LIN {X 62.159,Y -33.532,Z -240.496,A -90.000,B 90.000,C 0.000} C_DIS
LIN {X 62.499,Y -33.475,Z -240.051,A -90.000,B 90.000,C 0.000} C_DIS
LIN {X 62.795,Y -33.423,Z -239.682,A -90.000,B 90.000,C 0.000} C_DIS
LIN {X 62.961,Y -33.392,Z -239.489,A -90.000,B 90.000,C 0.000} C_DIS
LIN {X 63.098,Y -33.365,Z -239.345,A -90.000,B 90.000,C 0.000} C_DIS
LIN {X 63.154,Y -33.353,Z -239.294,A -90.000,B 90.000,C 0.000} C_DIS
LIN {X 63.202,Y -33.342,Z -239.257,A -90.000,B 90.000,C 0.000} C_DIS
LIN {X 63.241,Y -33.332,Z -239.236,A -90.000,B 90.000,C 0.000} C_DIS
LIN {X 63.256,Y -33.327,Z -239.231,A -90.000,B 90.000,C 0.000} C_DIS
LIN {X 63.276,Y -33.321,Z -239.232,A -90.000,B 90.000,C 0.000} C_DIS
LIN {X 63.285,Y -33.317,Z -239.238,A -90.000,B 90.000,C 0.000} C_DIS
LIN {X 63.295,Y -33.312,Z -239.255,A -90.000,B 90.000,C 0.000} C_DIS
LIN {X 63.298,Y -33.309,Z -239.272,A -90.000,B 90.000,C 0.000} C_DIS
LIN {X 63.296,Y -33.304,Z -239.320,A -90.000,B 90.000,C 0.000} C_DIS
LIN {X 63.282,Y -33.300,Z -239.387,A -90.000,B 90.000,C 0.000} C_DIS
LIN {X 63.240,Y -33.297,Z -239.526,A -90.000,B 90.000,C 0.000} C_DIS
LIN {X 63.169,Y -33.297,Z -239.713,A -90.000,B 90.000,C 0.000} C_DIS
LIN {X 63.030,Y -33.303,Z -240.041,A -90.000,B 90.000,C 0.000} C_DIS
LIN {X 62.938,Y -33.308,Z -240.240,A -90.000,B 90.000,C 0.000} C_DIS
LIN {X 62.258,Y -33.352,Z -241.702,A -90.000,B 90.000,C 0.000} C_DIS
LIN {X 61.796,Y -33.381,Z -242.689,A -90.000,B 90.000,C 0.000} C_DIS
LIN {X 61.390,Y -33.407,Z -243.561,A -90.000,B 90.000,C 0.000} C_DIS
LIN {X 61.390,Y -60.000,Z -243.561,A -90.000,B 90.000,C 0.000} C_DIS
LIN {X -95.002,Y -60.000,Z -243.561,A -90.000,B 90.000,C 0.000} C_DIS
LIN {X -95.002,Y -34.381,Z -243.561,A -90.000,B 90.000,C 0.000} C_DIS
LIN {X -94.873,Y -34.209,Z -243.260,A -90.000,B 90.000,C 0.000} C_DIS
LIN {X -94.532,Y -34.009,Z -242.776,A -90.000,B 90.000,C 0.000} C_DIS
LIN {X -94.065,Y -33.940,Z -242.365,A -90.000,B 90.000,C 0.000} C_DIS
LIN {X -92.639,Y -33.943,Z -241.367,A -90.000,B 90.000,C 0.000} C_DIS
LIN {X -91.606,Y -33.947,Z -240.642,A -90.000,B 90.000,C 0.000} C_DIS
LIN {X -89.459,Y -33.962,Z -239.147,A -90.000,B 90.000,C 0.000} C_DIS
LIN {X -88.994,Y -33.961,Z -238.830,A -90.000,B 90.000,C 0.000} C_DIS
LIN {X -88.572,Y -33.954,Z -238.548,A -90.000,B 90.000,C 0.000} C_DIS
LIN {X -88.341,Y -33.953,Z -238.396,A -90.000,B 90.000,C 0.000} C_DIS
LIN {X -86.770,Y -33.961,Z -237.376,A -90.000,B 90.000,C 0.000} C_DIS
LIN {X -84.189,Y -33.978,Z -235.700,A -90.000,B 90.000,C 0.000} C_DIS
LIN {X -80.955,Y -34.007,Z -233.615,A -90.000,B 90.000,C 0.000} C_DIS
LIN {X -80.422,Y -34.000,Z -233.284,A -90.000,B 90.000,C 0.000} C_DIS
LIN {X -80.197,Y -33.999,Z -233.147,A -90.000,B 90.000,C 0.000} C_DIS
LIN {X -78.206,Y -34.013,Z -231.959,A -90.000,B 90.000,C 0.000} C_DIS
LIN {X -73.699,Y -34.021,Z -229.309,A -90.000,B 90.000,C 0.000} C_DIS
LIN {X -72.528,Y -34.021,Z -228.623,A -90.000,B 90.000,C 0.000} C_DIS
LIN {X -71.738,Y -34.005,Z -228.177,A -90.000,B 90.000,C 0.000} C_DIS
LIN {X -67.969,Y -34.009,Z -226.154,A -90.000,B 90.000,C 0.000} C_DIS
LIN {X -63.803,Y -34.034,Z -223.947,A -90.000,B 90.000,C 0.000} C_DIS
LIN {X -63.185,Y -34.031,Z -223.626,A -90.000,B 90.000,C 0.000} C_DIS
LIN {X -62.836,Y -34.031,Z -223.448,A -90.000,B 90.000,C 0.000} C_DIS
LIN {X -59.942,Y -34.041,Z -221.989,A -90.000,B 90.000,C 0.000} C_DIS
LIN {X -54.944,Y -34.068,Z -219.481,A -90.000,B 90.000,C 0.000} C_DIS
LIN {X -54.352,Y -34.068,Z -219.187,A -90.000,B 90.000,C 0.000} C_DIS
LIN {X -49.979,Y -34.063,Z -217.035,A -90.000,B 90.000,C 0.000} C_DIS
LIN {X -47.190,Y -34.055,Z -215.668,A -90.000,B 90.000,C 0.000} C_DIS
LIN {X -46.482,Y -34.058,Z -215.318,A -90.000,B 90.000,C 0.000} C_DIS
LIN {X -45.806,Y -34.059,Z -214.980,A -90.000,B 90.000,C 0.000} C_DIS
LIN {X -40.274,Y -34.054,Z -212.247,A -90.000,B 90.000,C 0.000} C_DIS
LIN {X -39.897,Y -34.058,Z -212.057,A -90.000,B 90.000,C 0.000} C_DIS
LIN {X -39.523,Y -34.062,Z -211.867,A -90.000,B 90.000,C 0.000} C_DIS
LIN {X -38.424,Y -34.062,Z -211.295,A -90.000,B 90.000,C 0.000} C_DIS
LIN {X -36.891,Y -34.071,Z -210.490,A -90.000,B 90.000,C 0.000} C_DIS
LIN {X -34.601,Y -34.072,Z -209.269,A -90.000,B 90.000,C 0.000} C_DIS
LIN {X -34.129,Y -34.079,Z -209.011,A -90.000,B 90.000,C 0.000} C_DIS
LIN {X -32.795,Y -34.085,Z -208.262,A -90.000,B 90.000,C 0.000} C_DIS
LIN {X -30.542,Y -34.086,Z -206.982,A -90.000,B 90.000,C 0.000} C_DIS
LIN {X -29.946,Y -34.084,Z -206.646,A -90.000,B 90.000,C 0.000} C_DIS
LIN {X -29.328,Y -34.092,Z -206.286,A -90.000,B 90.000,C 0.000} C_DIS
LIN {X -28.104,Y -34.089,Z -205.541,A -90.000,B 90.000,C 0.000} C_DIS
LIN {X -26.597,Y -34.092,Z -204.635,A -90.000,B 90.000,C 0.000} C_DIS
LIN {X -25.789,Y -34.096,Z -204.147,A -90.000,B 90.000,C 0.000} C_DIS
LIN {X -25.670,Y -34.100,Z -204.073,A -90.000,B 90.000,C 0.000} C_DIS
LIN {X -25.200,Y -34.108,Z -203.778,A -90.000,B 90.000,C 0.000} C_DIS
LIN {X -23.362,Y -34.109,Z -202.572,A -90.000,B 90.000,C 0.000} C_DIS
LIN {X -22.534,Y -34.113,Z -202.026,A -90.000,B 90.000,C 0.000} C_DIS
LIN {X -22.232,Y -34.113,Z -201.824,A -90.000,B 90.000,C 0.000} C_DIS
LIN {X -21.655,Y -34.125,Z -201.428,A -90.000,B 90.000,C 0.000} C_DIS
LIN {X -20.573,Y -34.123,Z -200.645,A -90.000,B 90.000,C 0.000} C_DIS
LIN {X -20.238,Y -34.121,Z -200.404,A -90.000,B 90.000,C 0.000} C_DIS
LIN {X -18.840,Y -34.117,Z -199.408,A -90.000,B 90.000,C 0.000} C_DIS
LIN {X -18.234,Y -34.130,Z -198.963,A -90.000,B 90.000,C 0.000} C_DIS
LIN {X -16.865,Y -34.126,Z -197.899,A -90.000,B 90.000,C 0.000} C_DIS
LIN {X -16.453,Y -34.122,Z -197.581,A -90.000,B 90.000,C 0.000} C_DIS
LIN {X -15.403,Y -34.118,Z -196.780,A -90.000,B 90.000,C 0.000} C_DIS
LIN {X -14.781,Y -34.129,Z -196.292,A -90.000,B 90.000,C 0.000} C_DIS
LIN {X -13.118,Y -34.122,Z -194.933,A -90.000,B 90.000,C 0.000} C_DIS
LIN {X -12.741,Y -34.119,Z -194.626,A -90.000,B 90.000,C 0.000} C_DIS
LIN {X -11.964,Y -34.116,Z -194.000,A -90.000,B 90.000,C 0.000} C_DIS
LIN {X -11.322,Y -34.124,Z -193.473,A -90.000,B 90.000,C 0.000} C_DIS
LIN {X -9.514,Y -34.119,Z -191.943,A -90.000,B 90.000,C 0.000} C_DIS
LIN {X -8.977,Y -34.116,Z -191.491,A -90.000,B 90.000,C 0.000} C_DIS
LIN {X -8.420,Y -34.115,Z -191.025,A -90.000,B 90.000,C 0.000} C_DIS
LIN {X -7.757,Y -34.120,Z -190.465,A -90.000,B 90.000,C 0.000} C_DIS
LIN {X -6.654,Y -34.123,Z -189.524,A -90.000,B 90.000,C 0.000} C_DIS
LIN {X -4.663,Y -34.119,Z -187.811,A -90.000,B 90.000,C 0.000} C_DIS
LIN {X -3.934,Y -34.125,Z -187.175,A -90.000,B 90.000,C 0.000} C_DIS
LIN {X -3.262,Y -34.127,Z -186.589,A -90.000,B 90.000,C 0.000} C_DIS
LIN {X -0.962,Y -34.125,Z -184.573,A -90.000,B 90.000,C 0.000} C_DIS
LIN {X -0.258,Y -34.133,Z -183.947,A -90.000,B 90.000,C 0.000} C_DIS
LIN {X 2.548,Y -34.137,Z -181.427,A -90.000,B 90.000,C 0.000} C_DIS
LIN {X 3.185,Y -34.147,Z -180.848,A -90.000,B 90.000,C 0.000} C_DIS
LIN {X 5.800,Y -34.161,Z -178.421,A -90.000,B 90.000,C 0.000} C_DIS
LIN {X 6.267,Y -34.177,Z -177.976,A -90.000,B 90.000,C 0.000} C_DIS
LIN {X 6.719,Y -34.181,Z -177.529,A -90.000,B 90.000,C 0.000} C_DIS
LIN {X 8.383,Y -34.201,Z -175.896,A -90.000,B 90.000,C 0.000} C_DIS
LIN {X 8.757,Y -34.227,Z -175.511,A -90.000,B 90.000,C 0.000} C_DIS
LIN {X 8.969,Y -34.232,Z -175.270,A -90.000,B 90.000,C 0.000} C_DIS
LIN {X 9.243,Y -34.233,Z -174.965,A -90.000,B 90.000,C 0.000} C_DIS
LIN {X 10.634,Y -34.265,Z -173.481,A -90.000,B 90.000,C 0.000} C_DIS
LIN {X 10.935,Y -34.295,Z -173.139,A -90.000,B 90.000,C 0.000} C_DIS
LIN {X 11.307,Y -34.310,Z -172.649,A -90.000,B 90.000,C 0.000} C_DIS
LIN {X 11.613,Y -34.316,Z -172.255,A -90.000,B 90.000,C 0.000} C_DIS
LIN {X 12.194,Y -34.339,Z -171.552,A -90.000,B 90.000,C 0.000} C_DIS
LIN {X 12.454,Y -34.350,Z -171.236,A -90.000,B 90.000,C 0.000} C_DIS
LIN {X 12.590,Y -34.369,Z -171.060,A -90.000,B 90.000,C 0.000} C_DIS
LIN {X 13.208,Y -34.409,Z -170.063,A -90.000,B 90.000,C 0.000} C_DIS
LIN {X 13.528,Y -34.441,Z -169.537,A -90.000,B 90.000,C 0.000} C_DIS
LIN {X 13.656,Y -34.454,Z -169.331,A -90.000,B 90.000,C 0.000} C_DIS
LIN {X 13.733,Y -34.447,Z -169.124,A -90.000,B 90.000,C 0.000} C_DIS
LIN {X 13.863,Y -34.466,Z -168.731,A -90.000,B 90.000,C 0.000} C_DIS
LIN {X 14.347,Y -34.546,Z -167.346,A -90.000,B 90.000,C 0.000} C_DIS
LIN {X 14.354,Y -34.535,Z -167.206,A -90.000,B 90.000,C 0.000} C_DIS
LIN {X 14.359,Y -34.530,Z -166.963,A -90.000,B 90.000,C 0.000} C_DIS
LIN {X 14.381,Y -34.522,Z -166.386,A -90.000,B 90.000,C 0.000} C_DIS
LIN {X 14.385,Y -34.535,Z -166.076,A -90.000,B 90.000,C 0.000} C_DIS
LIN {X 14.323,Y -34.519,Z -165.696,A -90.000,B 90.000,C 0.000} C_DIS
LIN {X 14.225,Y -34.499,Z -165.096,A -90.000,B 90.000,C 0.000} C_DIS
LIN {X 14.177,Y -34.494,Z -164.732,A -90.000,B 90.000,C 0.000} C_DIS
LIN {X 14.159,Y -34.492,Z -164.583,A -90.000,B 90.000,C 0.000} C_DIS
LIN {X 14.148,Y -34.496,Z -164.509,A -90.000,B 90.000,C 0.000} C_DIS
LIN {X 14.005,Y -34.503,Z -163.900,A -90.000,B 90.000,C 0.000} C_DIS
LIN {X 13.939,Y -34.502,Z -163.607,A -90.000,B 90.000,C 0.000} C_DIS
LIN {X 13.827,Y -34.477,Z -163.300,A -90.000,B 90.000,C 0.000} C_DIS
LIN {X 13.788,Y -34.474,Z -163.199,A -90.000,B 90.000,C 0.000} C_DIS
LIN {X 13.731,Y -34.472,Z -163.029,A -90.000,B 90.000,C 0.000} C_DIS
LIN {X 13.487,Y -34.477,Z -162.191,A -90.000,B 90.000,C 0.000} C_DIS
LIN {X 13.390,Y -34.468,Z -161.928,A -90.000,B 90.000,C 0.000} C_DIS
LIN {X 13.165,Y -34.469,Z -161.344,A -90.000,B 90.000,C 0.000} C_DIS
LIN {X 12.973,Y -34.468,Z -160.825,A -90.000,B 90.000,C 0.000} C_DIS
LIN {X 12.829,Y -34.465,Z -160.458,A -90.000,B 90.000,C 0.000} C_DIS
LIN {X 12.638,Y -34.483,Z -159.999,A -90.000,B 90.000,C 0.000} C_DIS
LIN {X 12.561,Y -34.483,Z -159.848,A -90.000,B 90.000,C 0.000} C_DIS
LIN {X 12.508,Y -34.485,Z -159.739,A -90.000,B 90.000,C 0.000} C_DIS
LIN {X 12.231,Y -34.502,Z -159.117,A -90.000,B 90.000,C 0.000} C_DIS
LIN {X 12.053,Y -34.502,Z -158.705,A -90.000,B 90.000,C 0.000} C_DIS
LIN {X 11.900,Y -34.534,Z -158.371,A -90.000,B 90.000,C 0.000} C_DIS
LIN {X 11.754,Y -34.550,Z -158.111,A -90.000,B 90.000,C 0.000} C_DIS
LIN {X 11.569,Y -34.577,Z -157.758,A -90.000,B 90.000,C 0.000} C_DIS
LIN {X 11.396,Y -34.594,Z -157.422,A -90.000,B 90.000,C 0.000} C_DIS
LIN {X 11.280,Y -34.597,Z -157.187,A -90.000,B 90.000,C 0.000} C_DIS
LIN {X 11.173,Y -34.599,Z -156.961,A -90.000,B 90.000,C 0.000} C_DIS
LIN {X 10.963,Y -34.659,Z -156.564,A -90.000,B 90.000,C 0.000} C_DIS
LIN {X 10.916,Y -34.674,Z -156.471,A -90.000,B 90.000,C 0.000} C_DIS
LIN {X 10.594,Y -34.723,Z -156.014,A -90.000,B 90.000,C 0.000} C_DIS
LIN {X 10.530,Y -34.725,Z -155.919,A -90.000,B 90.000,C 0.000} C_DIS
LIN {X 10.447,Y -34.729,Z -155.796,A -90.000,B 90.000,C 0.000} C_DIS
LIN {X 10.355,Y -34.729,Z -155.658,A -90.000,B 90.000,C 0.000} C_DIS
LIN {X 10.137,Y -34.703,Z -155.488,A -90.000,B 90.000,C 0.000} C_DIS
LIN {X 10.023,Y -34.711,Z -155.408,A -90.000,B 90.000,C 0.000} C_DIS
LIN {X 9.378,Y -34.642,Z -155.286,A -90.000,B 90.000,C 0.000} C_DIS
LIN {X 9.325,Y -34.633,Z -155.286,A -90.000,B 90.000,C 0.000} C_DIS
LIN {X 8.705,Y -34.516,Z -155.315,A -90.000,B 90.000,C 0.000} C_DIS
LIN {X 8.296,Y -34.437,Z -155.335,A -90.000,B 90.000,C 0.000} C_DIS
LIN {X 8.001,Y -34.381,Z -155.347,A -90.000,B 90.000,C 0.000} C_DIS
LIN {X 7.415,Y -34.271,Z -155.366,A -90.000,B 90.000,C 0.000} C_DIS
LIN {X 7.286,Y -34.249,Z -155.365,A -90.000,B 90.000,C 0.000} C_DIS
LIN {X 6.859,Y -34.180,Z -155.350,A -90.000,B 90.000,C 0.000} C_DIS
LIN {X 6.747,Y -34.168,Z -155.347,A -90.000,B 90.000,C 0.000} C_DIS
LIN {X 5.769,Y -34.082,Z -155.287,A -90.000,B 90.000,C 0.000} C_DIS
LIN {X 4.976,Y -34.004,Z -155.251,A -90.000,B 90.000,C 0.000} C_DIS
LIN {X 4.684,Y -33.973,Z -155.233,A -90.000,B 90.000,C 0.000} C_DIS
LIN {X 3.965,Y -33.883,Z -155.172,A -90.000,B 90.000,C 0.000} C_DIS
LIN {X 3.466,Y -33.830,Z -155.115,A -90.000,B 90.000,C 0.000} C_DIS
LIN {X 3.329,Y -33.819,Z -155.094,A -90.000,B 90.000,C 0.000} C_DIS
LIN {X 3.084,Y -33.803,Z -155.049,A -90.000,B 90.000,C 0.000} C_DIS
LIN {X 2.395,Y -33.753,Z -154.935,A -90.000,B 90.000,C 0.000} C_DIS
LIN {X 2.021,Y -33.726,Z -154.871,A -90.000,B 90.000,C 0.000} C_DIS
LIN {X 0.609,Y -33.706,Z -154.731,A -90.000,B 90.000,C 0.000} C_DIS
LIN {X 0.262,Y -33.693,Z -154.684,A -90.000,B 90.000,C 0.000} C_DIS
LIN {X 0.196,Y -33.691,Z -154.674,A -90.000,B 90.000,C 0.000} C_DIS
LIN {X 0.043,Y -33.679,Z -154.641,A -90.000,B 90.000,C 0.000} C_DIS
LIN {X -0.196,Y -33.664,Z -154.586,A -90.000,B 90.000,C 0.000} C_DIS
LIN {X -0.331,Y -33.657,Z -154.551,A -90.000,B 90.000,C 0.000} C_DIS
LIN {X -0.436,Y -33.651,Z -154.524,A -90.000,B 90.000,C 0.000} C_DIS
LIN {X -1.538,Y -33.604,Z -154.234,A -90.000,B 90.000,C 0.000} C_DIS
LIN {X -3.542,Y -33.575,Z -153.793,A -90.000,B 90.000,C 0.000} C_DIS
LIN {X -3.731,Y -33.568,Z -153.746,A -90.000,B 90.000,C 0.000} C_DIS
LIN {X -3.983,Y -33.567,Z -153.678,A -90.000,B 90.000,C 0.000} C_DIS
LIN {X -4.254,Y -33.557,Z -153.585,A -90.000,B 90.000,C 0.000} C_DIS
LIN {X -4.866,Y -33.542,Z -153.370,A -90.000,B 90.000,C 0.000} C_DIS
LIN {X -7.627,Y -33.508,Z -152.461,A -90.000,B 90.000,C 0.000} C_DIS
LIN {X -7.821,Y -33.503,Z -152.386,A -90.000,B 90.000,C 0.000} C_DIS
LIN {X -8.062,Y -33.503,Z -152.291,A -90.000,B 90.000,C 0.000} C_DIS
LIN {X -8.911,Y -33.490,Z -151.916,A -90.000,B 90.000,C 0.000} C_DIS
LIN {X -11.590,Y -33.475,Z -150.786,A -90.000,B 90.000,C 0.000} C_DIS
LIN {X -11.853,Y -33.469,Z -150.658,A -90.000,B 90.000,C 0.000} C_DIS
LIN {X -11.961,Y -33.469,Z -150.604,A -90.000,B 90.000,C 0.000} C_DIS
LIN {X -15.601,Y -33.463,Z -148.685,A -90.000,B 90.000,C 0.000} C_DIS
LIN {X -15.999,Y -33.450,Z -148.437,A -90.000,B 90.000,C 0.000} C_DIS
LIN {X -17.159,Y -33.450,Z -147.679,A -90.000,B 90.000,C 0.000} C_DIS
LIN {X -18.184,Y -33.448,Z -147.012,A -90.000,B 90.000,C 0.000} C_DIS
LIN {X -19.611,Y -33.452,Z -146.104,A -90.000,B 90.000,C 0.000} C_DIS
LIN {X -20.052,Y -33.440,Z -145.768,A -90.000,B 90.000,C 0.000} C_DIS
LIN {X -20.565,Y -33.442,Z -145.372,A -90.000,B 90.000,C 0.000} C_DIS
LIN {X -21.386,Y -33.451,Z -144.756,A -90.000,B 90.000,C 0.000} C_DIS
LIN {X -21.965,Y -33.458,Z -144.321,A -90.000,B 90.000,C 0.000} C_DIS
LIN {X -23.150,Y -33.462,Z -143.408,A -90.000,B 90.000,C 0.000} C_DIS
LIN {X -23.377,Y -33.461,Z -143.227,A -90.000,B 90.000,C 0.000} C_DIS
LIN {X -23.522,Y -33.459,Z -143.110,A -90.000,B 90.000,C 0.000} C_DIS
LIN {X -23.953,Y -33.451,Z -142.721,A -90.000,B 90.000,C 0.000} C_DIS
LIN {X -24.567,Y -33.453,Z -142.160,A -90.000,B 90.000,C 0.000} C_DIS
LIN {X -25.089,Y -33.453,Z -141.686,A -90.000,B 90.000,C 0.000} C_DIS
LIN {X -25.435,Y -33.455,Z -141.379,A -90.000,B 90.000,C 0.000} C_DIS
LIN {X -26.824,Y -33.470,Z -140.144,A -90.000,B 90.000,C 0.000} C_DIS
LIN {X -27.164,Y -33.466,Z -139.812,A -90.000,B 90.000,C 0.000} C_DIS
LIN {X -27.335,Y -33.467,Z -139.632,A -90.000,B 90.000,C 0.000} C_DIS
LIN {X -27.651,Y -33.467,Z -139.290,A -90.000,B 90.000,C 0.000} C_DIS
LIN {X -29.301,Y -33.483,Z -137.499,A -90.000,B 90.000,C 0.000} C_DIS
LIN {X -29.738,Y -33.485,Z -137.021,A -90.000,B 90.000,C 0.000} C_DIS
LIN {X -30.075,Y -33.489,Z -136.657,A -90.000,B 90.000,C 0.000} C_DIS
LIN {X -30.270,Y -33.483,Z -136.415,A -90.000,B 90.000,C 0.000} C_DIS
LIN {X -30.331,Y -33.484,Z -136.338,A -90.000,B 90.000,C 0.000} C_DIS
LIN {X -30.554,Y -33.484,Z -136.043,A -90.000,B 90.000,C 0.000} C_DIS
LIN {X -30.864,Y -33.488,Z -135.631,A -90.000,B 90.000,C 0.000} C_DIS
LIN {X -31.747,Y -33.500,Z -134.465,A -90.000,B 90.000,C 0.000} C_DIS
LIN {X -32.528,Y -33.510,Z -133.429,A -90.000,B 90.000,C 0.000} C_DIS
LIN {X -32.708,Y -33.515,Z -133.188,A -90.000,B 90.000,C 0.000} C_DIS
LIN {X -32.842,Y -33.513,Z -132.986,A -90.000,B 90.000,C 0.000} C_DIS
LIN {X -33.085,Y -33.515,Z -132.587,A -90.000,B 90.000,C 0.000} C_DIS
LIN {X -33.931,Y -33.537,Z -131.182,A -90.000,B 90.000,C 0.000} C_DIS
LIN {X -34.648,Y -33.548,Z -129.959,A -90.000,B 90.000,C 0.000} C_DIS
LIN {X -34.862,Y -33.553,Z -129.592,A -90.000,B 90.000,C 0.000} C_DIS
LIN {X -35.417,Y -33.562,Z -128.408,A -90.000,B 90.000,C 0.000} C_DIS
LIN {X -36.360,Y -33.581,Z -126.392,A -90.000,B 90.000,C 0.000} C_DIS
LIN {X -36.465,Y -33.583,Z -126.158,A -90.000,B 90.000,C 0.000} C_DIS
LIN {X -36.523,Y -33.588,Z -126.023,A -90.000,B 90.000,C 0.000} C_DIS
LIN {X -36.814,Y -33.590,Z -125.230,A -90.000,B 90.000,C 0.000} C_DIS
LIN {X -37.530,Y -33.594,Z -123.280,A -90.000,B 90.000,C 0.000} C_DIS
LIN {X -37.657,Y -33.600,Z -122.924,A -90.000,B 90.000,C 0.000} C_DIS
LIN {X -37.693,Y -33.601,Z -122.812,A -90.000,B 90.000,C 0.000} C_DIS
LIN {X -37.789,Y -33.607,Z -122.510,A -90.000,B 90.000,C 0.000} C_DIS
LIN {X -38.196,Y -33.590,Z -121.049,A -90.000,B 90.000,C 0.000} C_DIS
LIN {X -38.509,Y -33.587,Z -119.908,A -90.000,B 90.000,C 0.000} C_DIS
LIN {X -38.595,Y -33.596,Z -119.573,A -90.000,B 90.000,C 0.000} C_DIS
LIN {X -38.682,Y -33.602,Z -119.190,A -90.000,B 90.000,C 0.000} C_DIS
LIN {X -38.743,Y -33.601,Z -118.872,A -90.000,B 90.000,C 0.000} C_DIS
LIN {X -38.935,Y -33.593,Z -117.837,A -90.000,B 90.000,C 0.000} C_DIS
LIN {X -39.032,Y -33.587,Z -117.334,A -90.000,B 90.000,C 0.000} C_DIS
LIN {X -39.215,Y -33.579,Z -116.390,A -90.000,B 90.000,C 0.000} C_DIS
LIN {X -39.230,Y -33.580,Z -116.307,A -90.000,B 90.000,C 0.000} C_DIS
LIN {X -39.358,Y -33.602,Z -115.575,A -90.000,B 90.000,C 0.000} C_DIS
LIN {X -39.399,Y -33.596,Z -115.225,A -90.000,B 90.000,C 0.000} C_DIS
LIN {X -39.428,Y -33.592,Z -114.983,A -90.000,B 90.000,C 0.000} C_DIS
LIN {X -39.502,Y -33.578,Z -114.284,A -90.000,B 90.000,C 0.000} C_DIS
LIN {X -39.601,Y -33.570,Z -113.300,A -90.000,B 90.000,C 0.000} C_DIS
LIN {X -39.645,Y -33.571,Z -112.836,A -90.000,B 90.000,C 0.000} C_DIS
LIN {X -39.674,Y -33.580,Z -112.458,A -90.000,B 90.000,C 0.000} C_DIS
LIN {X -39.696,Y -33.590,Z -112.185,A -90.000,B 90.000,C 0.000} C_DIS
LIN {X -39.720,Y -33.600,Z -111.769,A -90.000,B 90.000,C 0.000} C_DIS
LIN {X -39.725,Y -33.597,Z -111.269,A -90.000,B 90.000,C 0.000} C_DIS
LIN {X -39.728,Y -33.593,Z -110.998,A -90.000,B 90.000,C 0.000} C_DIS
LIN {X -39.750,Y -33.583,Z -109.970,A -90.000,B 90.000,C 0.000} C_DIS
LIN {X -39.755,Y -33.578,Z -109.563,A -90.000,B 90.000,C 0.000} C_DIS
LIN {X -39.755,Y -33.584,Z -109.062,A -90.000,B 90.000,C 0.000} C_DIS
LIN {X -39.755,Y -33.585,Z -109.015,A -90.000,B 90.000,C 0.000} C_DIS
LIN {X -39.752,Y -33.601,Z -108.594,A -90.000,B 90.000,C 0.000} C_DIS
LIN {X -39.738,Y -33.617,Z -108.151,A -90.000,B 90.000,C 0.000} C_DIS
LIN {X -39.618,Y -33.621,Z -106.728,A -90.000,B 90.000,C 0.000} C_DIS
LIN {X -39.591,Y -33.630,Z -106.282,A -90.000,B 90.000,C 0.000} C_DIS
LIN {X -39.570,Y -33.641,Z -105.984,A -90.000,B 90.000,C 0.000} C_DIS
LIN {X -39.574,Y -33.649,Z -105.933,A -90.000,B 90.000,C 0.000} C_DIS
LIN {X -39.603,Y -33.689,Z -105.733,A -90.000,B 90.000,C 0.000} C_DIS
LIN {X -39.687,Y -33.905,Z -104.786,A -90.000,B 90.000,C 0.000} C_DIS
LIN {X -39.703,Y -33.985,Z -104.461,A -90.000,B 90.000,C 0.000} C_DIS
LIN {X -39.715,Y -34.034,Z -104.290,A -90.000,B 90.000,C 0.000} C_DIS
LIN {X -39.730,Y -34.114,Z -104.019,A -90.000,B 90.000,C 0.000} C_DIS
LIN {X -39.737,Y -34.256,Z -103.511,A -90.000,B 90.000,C 0.000} C_DIS
LIN {X -39.735,Y -34.336,Z -103.233,A -90.000,B 90.000,C 0.000} C_DIS
LIN {X -39.728,Y -34.377,Z -103.097,A -90.000,B 90.000,C 0.000} C_DIS
LIN {X -39.716,Y -34.428,Z -102.932,A -90.000,B 90.000,C 0.000} C_DIS
LIN {X -39.687,Y -34.522,Z -102.629,A -90.000,B 90.000,C 0.000} C_DIS
LIN {X -39.794,Y -34.529,Z -102.461,A -90.000,B 90.000,C 0.000} C_DIS
LIN {X -39.978,Y -34.527,Z -102.218,A -90.000,B 90.000,C 0.000} C_DIS
LIN {X -40.274,Y -34.520,Z -101.825,A -90.000,B 90.000,C 0.000} C_DIS
LIN {X -40.484,Y -34.518,Z -101.540,A -90.000,B 90.000,C 0.000} C_DIS
LIN {X -40.926,Y -34.522,Z -100.945,A -90.000,B 90.000,C 0.000} C_DIS
LIN {X -41.149,Y -34.528,Z -100.633,A -90.000,B 90.000,C 0.000} C_DIS
LIN {X -41.594,Y -34.528,Z -99.995,A -90.000,B 90.000,C 0.000} C_DIS
LIN {X -41.989,Y -34.521,Z -99.424,A -90.000,B 90.000,C 0.000} C_DIS
LIN {X -42.209,Y -34.519,Z -99.094,A -90.000,B 90.000,C 0.000} C_DIS
LIN {X -43.182,Y -34.537,Z -97.528,A -90.000,B 90.000,C 0.000} C_DIS
LIN {X -43.779,Y -34.537,Z -96.531,A -90.000,B 90.000,C 0.000} C_DIS
LIN {X -44.127,Y -34.542,Z -95.910,A -90.000,B 90.000,C 0.000} C_DIS
LIN {X -44.243,Y -34.545,Z -95.693,A -90.000,B 90.000,C 0.000} C_DIS
LIN {X -44.690,Y -34.548,Z -94.867,A -90.000,B 90.000,C 0.000} C_DIS
LIN {X -45.006,Y -34.543,Z -94.279,A -90.000,B 90.000,C 0.000} C_DIS
LIN {X -45.634,Y -34.529,Z -93.045,A -90.000,B 90.000,C 0.000} C_DIS
LIN {X -45.784,Y -34.527,Z -92.725,A -90.000,B 90.000,C 0.000} C_DIS
LIN {X -45.928,Y -34.524,Z -92.409,A -90.000,B 90.000,C 0.000} C_DIS
LIN {X -46.226,Y -34.527,Z -91.706,A -90.000,B 90.000,C 0.000} C_DIS
LIN {X -46.345,Y -34.531,Z -91.429,A -90.000,B 90.000,C 0.000} C_DIS
LIN {X -46.588,Y -34.531,Z -90.852,A -90.000,B 90.000,C 0.000} C_DIS
LIN {X -46.672,Y -34.529,Z -90.650,A -90.000,B 90.000,C 0.000} C_DIS
LIN {X -46.795,Y -34.524,Z -90.342,A -90.000,B 90.000,C 0.000} C_DIS
LIN {X -47.062,Y -34.518,Z -89.640,A -90.000,B 90.000,C 0.000} C_DIS
LIN {X -47.276,Y -34.515,Z -89.066,A -90.000,B 90.000,C 0.000} C_DIS
LIN {X -47.307,Y -34.515,Z -88.976,A -90.000,B 90.000,C 0.000} C_DIS
LIN {X -47.481,Y -34.521,Z -88.439,A -90.000,B 90.000,C 0.000} C_DIS
LIN {X -47.708,Y -34.530,Z -87.635,A -90.000,B 90.000,C 0.000} C_DIS
LIN {X -47.958,Y -34.555,Z -86.619,A -90.000,B 90.000,C 0.000} C_DIS
LIN {X -48.119,Y -34.563,Z -85.944,A -90.000,B 90.000,C 0.000} C_DIS
LIN {X -48.237,Y -34.565,Z -85.444,A -90.000,B 90.000,C 0.000} C_DIS
LIN {X -48.290,Y -34.565,Z -85.230,A -90.000,B 90.000,C 0.000} C_DIS
LIN {X -48.318,Y -34.563,Z -85.110,A -90.000,B 90.000,C 0.000} C_DIS
LIN {X -48.354,Y -34.562,Z -84.920,A -90.000,B 90.000,C 0.000} C_DIS
LIN {X -48.399,Y -34.567,Z -84.609,A -90.000,B 90.000,C 0.000} C_DIS
LIN {X -48.445,Y -34.574,Z -84.247,A -90.000,B 90.000,C 0.000} C_DIS
LIN {X -48.490,Y -34.586,Z -83.828,A -90.000,B 90.000,C 0.000} C_DIS
LIN {X -48.573,Y -34.613,Z -83.086,A -90.000,B 90.000,C 0.000} C_DIS
LIN {X -48.605,Y -34.616,Z -82.769,A -90.000,B 90.000,C 0.000} C_DIS
LIN {X -48.642,Y -34.615,Z -82.371,A -90.000,B 90.000,C 0.000} C_DIS
LIN {X -48.646,Y -34.620,Z -82.172,A -90.000,B 90.000,C 0.000} C_DIS
LIN {X -48.616,Y -34.663,Z -81.147,A -90.000,B 90.000,C 0.000} C_DIS
LIN {X -48.606,Y -34.674,Z -80.924,A -90.000,B 90.000,C 0.000} C_DIS
LIN {X -48.552,Y -34.680,Z -79.949,A -90.000,B 90.000,C 0.000} C_DIS
LIN {X -48.532,Y -34.685,Z -79.752,A -90.000,B 90.000,C 0.000} C_DIS
LIN {X -48.441,Y -34.707,Z -79.153,A -90.000,B 90.000,C 0.000} C_DIS
LIN {X -48.394,Y -34.717,Z -78.846,A -90.000,B 90.000,C 0.000} C_DIS
LIN {X -48.360,Y -34.721,Z -78.650,A -90.000,B 90.000,C 0.000} C_DIS
LIN {X -48.232,Y -34.730,Z -77.986,A -90.000,B 90.000,C 0.000} C_DIS
LIN {X -48.159,Y -34.735,Z -77.625,A -90.000,B 90.000,C 0.000} C_DIS
LIN {X -48.134,Y -34.738,Z -77.513,A -90.000,B 90.000,C 0.000} C_DIS
LIN {X -47.991,Y -34.754,Z -76.959,A -90.000,B 90.000,C 0.000} C_DIS
LIN {X -47.818,Y -34.767,Z -76.298,A -90.000,B 90.000,C 0.000} C_DIS
LIN {X -47.774,Y -34.768,Z -76.136,A -90.000,B 90.000,C 0.000} C_DIS
LIN {X -47.689,Y -34.771,Z -75.857,A -90.000,B 90.000,C 0.000} C_DIS
LIN {X -47.567,Y -34.777,Z -75.486,A -90.000,B 90.000,C 0.000} C_DIS
LIN {X -47.263,Y -34.794,Z -74.623,A -90.000,B 90.000,C 0.000} C_DIS
LIN {X -47.123,Y -34.795,Z -74.230,A -90.000,B 90.000,C 0.000} C_DIS
LIN {X -47.075,Y -34.796,Z -74.107,A -90.000,B 90.000,C 0.000} C_DIS
LIN {X -46.850,Y -34.804,Z -73.585,A -90.000,B 90.000,C 0.000} C_DIS
LIN {X -46.642,Y -34.812,Z -73.094,A -90.000,B 90.000,C 0.000} C_DIS
LIN {X -46.444,Y -34.811,Z -72.632,A -90.000,B 90.000,C 0.000} C_DIS
LIN {X -46.371,Y -34.812,Z -72.477,A -90.000,B 90.000,C 0.000} C_DIS
LIN {X -46.171,Y -34.817,Z -72.066,A -90.000,B 90.000,C 0.000} C_DIS
LIN {X -46.140,Y -34.816,Z -72.004,A -90.000,B 90.000,C 0.000} C_DIS
LIN {X -45.985,Y -34.817,Z -71.720,A -90.000,B 90.000,C 0.000} C_DIS
LIN {X -45.865,Y -34.818,Z -71.518,A -90.000,B 90.000,C 0.000} C_DIS
LIN {X -45.457,Y -34.816,Z -70.840,A -90.000,B 90.000,C 0.000} C_DIS
LIN {X -45.413,Y -34.817,Z -70.771,A -90.000,B 90.000,C 0.000} C_DIS
LIN {X -45.178,Y -34.820,Z -70.412,A -90.000,B 90.000,C 0.000} C_DIS
LIN {X -44.948,Y -34.806,Z -70.070,A -90.000,B 90.000,C 0.000} C_DIS
LIN {X -44.890,Y -34.803,Z -69.989,A -90.000,B 90.000,C 0.000} C_DIS
LIN {X -44.795,Y -34.800,Z -69.873,A -90.000,B 90.000,C 0.000} C_DIS
LIN {X -44.594,Y -34.796,Z -69.646,A -90.000,B 90.000,C 0.000} C_DIS
LIN {X -44.093,Y -34.796,Z -69.111,A -90.000,B 90.000,C 0.000} C_DIS
LIN {X -43.839,Y -34.796,Z -68.858,A -90.000,B 90.000,C 0.000} C_DIS
LIN {X -43.669,Y -34.786,Z -68.693,A -90.000,B 90.000,C 0.000} C_DIS
LIN {X -43.172,Y -34.748,Z -68.214,A -90.000,B 90.000,C 0.000} C_DIS
LIN {X -42.967,Y -34.737,Z -68.041,A -90.000,B 90.000,C 0.000} C_DIS
LIN {X -42.872,Y -34.735,Z -67.971,A -90.000,B 90.000,C 0.000} C_DIS
LIN {X -42.746,Y -34.732,Z -67.878,A -90.000,B 90.000,C 0.000} C_DIS
LIN {X -42.462,Y -34.726,Z -67.688,A -90.000,B 90.000,C 0.000} C_DIS
LIN {X -42.330,Y -34.725,Z -67.607,A -90.000,B 90.000,C 0.000} C_DIS
LIN {X -41.755,Y -34.730,Z -67.283,A -90.000,B 90.000,C 0.000} C_DIS
LIN {X -41.518,Y -34.726,Z -67.152,A -90.000,B 90.000,C 0.000} C_DIS
LIN {X -41.075,Y -34.691,Z -66.916,A -90.000,B 90.000,C 0.000} C_DIS
LIN {X -41.005,Y -34.686,Z -66.880,A -90.000,B 90.000,C 0.000} C_DIS
LIN {X -40.436,Y -34.650,Z -66.605,A -90.000,B 90.000,C 0.000} C_DIS
LIN {X -39.679,Y -34.590,Z -66.246,A -90.000,B 90.000,C 0.000} C_DIS
LIN {X -39.407,Y -34.578,Z -66.146,A -90.000,B 90.000,C 0.000} C_DIS
LIN {X -39.065,Y -34.574,Z -66.047,A -90.000,B 90.000,C 0.000} C_DIS
LIN {X -38.940,Y -34.574,Z -66.015,A -90.000,B 90.000,C 0.000} C_DIS
LIN {X -38.037,Y -34.559,Z -65.791,A -90.000,B 90.000,C 0.000} C_DIS
LIN {X -37.932,Y -34.556,Z -65.771,A -90.000,B 90.000,C 0.000} C_DIS
LIN {X -37.272,Y -34.543,Z -65.663,A -90.000,B 90.000,C 0.000} C_DIS
LIN {X -36.781,Y -34.522,Z -65.587,A -90.000,B 90.000,C 0.000} C_DIS
LIN {X -36.695,Y -34.519,Z -65.576,A -90.000,B 90.000,C 0.000} C_DIS
LIN {X -35.629,Y -34.489,Z -65.457,A -90.000,B 90.000,C 0.000} C_DIS
LIN {X -34.818,Y -34.447,Z -65.376,A -90.000,B 90.000,C 0.000} C_DIS
LIN {X -34.628,Y -34.438,Z -65.359,A -90.000,B 90.000,C 0.000} C_DIS
LIN {X -34.496,Y -34.434,Z -65.351,A -90.000,B 90.000,C 0.000} C_DIS
LIN {X -34.409,Y -34.432,Z -65.348,A -90.000,B 90.000,C 0.000} C_DIS
LIN {X -34.053,Y -34.430,Z -65.343,A -90.000,B 90.000,C 0.000} C_DIS
LIN {X -33.789,Y -34.424,Z -65.341,A -90.000,B 90.000,C 0.000} C_DIS
LIN {X -32.580,Y -34.374,Z -65.348,A -90.000,B 90.000,C 0.000} C_DIS
LIN {X -31.926,Y -34.362,Z -65.380,A -90.000,B 90.000,C 0.000} C_DIS
LIN {X -31.370,Y -34.363,Z -65.428,A -90.000,B 90.000,C 0.000} C_DIS
LIN {X -31.067,Y -34.367,Z -65.462,A -90.000,B 90.000,C 0.000} C_DIS
LIN {X -30.780,Y -34.362,Z -65.500,A -90.000,B 90.000,C 0.000} C_DIS
LIN {X -29.591,Y -34.331,Z -65.662,A -90.000,B 90.000,C 0.000} C_DIS
LIN {X -29.080,Y -34.320,Z -65.737,A -90.000,B 90.000,C 0.000} C_DIS
LIN {X -28.944,Y -34.318,Z -65.762,A -90.000,B 90.000,C 0.000} C_DIS
LIN {X -28.463,Y -34.318,Z -65.861,A -90.000,B 90.000,C 0.000} C_DIS
LIN {X -27.096,Y -34.294,Z -66.159,A -90.000,B 90.000,C 0.000} C_DIS
LIN {X -26.948,Y -34.293,Z -66.194,A -90.000,B 90.000,C 0.000} C_DIS
LIN {X -26.416,Y -34.289,Z -66.319,A -90.000,B 90.000,C 0.000} C_DIS
LIN {X -24.780,Y -34.272,Z -66.817,A -90.000,B 90.000,C 0.000} C_DIS
LIN {X -24.466,Y -34.271,Z -66.918,A -90.000,B 90.000,C 0.000} C_DIS
LIN {X -24.206,Y -34.272,Z -67.005,A -90.000,B 90.000,C 0.000} C_DIS
LIN {X -23.079,Y -34.262,Z -67.388,A -90.000,B 90.000,C 0.000} C_DIS
LIN {X -22.862,Y -34.263,Z -67.465,A -90.000,B 90.000,C 0.000} C_DIS
LIN {X -22.752,Y -34.260,Z -67.499,A -90.000,B 90.000,C 0.000} C_DIS
LIN {X -21.748,Y -34.250,Z -67.803,A -90.000,B 90.000,C 0.000} C_DIS
LIN {X -21.646,Y -34.243,Z -67.822,A -90.000,B 90.000,C 0.000} C_DIS
LIN {X -21.567,Y -34.242,Z -67.835,A -90.000,B 90.000,C 0.000} C_DIS
LIN {X -21.207,Y -34.148,Z -67.758,A -90.000,B 90.000,C 0.000} C_DIS
LIN {X -20.990,Y -34.124,Z -67.685,A -90.000,B 90.000,C 0.000} C_DIS
LIN {X -20.929,Y -34.123,Z -67.659,A -90.000,B 90.000,C 0.000} C_DIS
LIN {X -20.656,Y -34.136,Z -67.536,A -90.000,B 90.000,C 0.000} C_DIS
LIN {X -20.223,Y -34.159,Z -67.348,A -90.000,B 90.000,C 0.000} C_DIS
LIN {X -20.166,Y -34.161,Z -67.323,A -90.000,B 90.000,C 0.000} C_DIS
LIN {X -20.009,Y -34.186,Z -67.244,A -90.000,B 90.000,C 0.000} C_DIS
LIN {X -19.675,Y -34.243,Z -67.086,A -90.000,B 90.000,C 0.000} C_DIS
LIN {X -19.517,Y -34.272,Z -67.019,A -90.000,B 90.000,C 0.000} C_DIS
LIN {X -19.376,Y -34.297,Z -66.969,A -90.000,B 90.000,C 0.000} C_DIS
LIN {X -19.328,Y -34.308,Z -66.951,A -90.000,B 90.000,C 0.000} C_DIS
LIN {X -18.683,Y -34.418,Z -66.729,A -90.000,B 90.000,C 0.000} C_DIS
LIN {X -18.285,Y -34.486,Z -66.596,A -90.000,B 90.000,C 0.000} C_DIS
LIN {X -18.156,Y -34.507,Z -66.547,A -90.000,B 90.000,C 0.000} C_DIS
LIN {X -17.840,Y -34.577,Z -66.420,A -90.000,B 90.000,C 0.000} C_DIS
LIN {X -17.715,Y -34.605,Z -66.376,A -90.000,B 90.000,C 0.000} C_DIS
LIN {X -17.306,Y -34.699,Z -66.257,A -90.000,B 90.000,C 0.000} C_DIS
LIN {X -17.229,Y -34.717,Z -66.238,A -90.000,B 90.000,C 0.000} C_DIS
LIN {X -16.755,Y -34.789,Z -66.158,A -90.000,B 90.000,C 0.000} C_DIS
LIN {X -16.701,Y -34.797,Z -66.149,A -90.000,B 90.000,C 0.000} C_DIS
LIN {X -16.000,Y -34.874,Z -66.044,A -90.000,B 90.000,C 0.000} C_DIS
LIN {X -15.267,Y -34.958,Z -65.955,A -90.000,B 90.000,C 0.000} C_DIS
LIN {X -14.703,Y -35.017,Z -65.801,A -90.000,B 90.000,C 0.000} C_DIS
LIN {X -14.435,Y -35.046,Z -65.748,A -90.000,B 90.000,C 0.000} C_DIS
LIN {X -14.143,Y -35.080,Z -65.712,A -90.000,B 90.000,C 0.000} C_DIS
LIN {X -13.949,Y -35.099,Z -65.647,A -90.000,B 90.000,C 0.000} C_DIS
LIN {X -13.779,Y -35.101,Z -65.480,A -90.000,B 90.000,C 0.000} C_DIS
LIN {X -13.649,Y -35.094,Z -65.354,A -90.000,B 90.000,C 0.000} C_DIS
LIN {X -13.575,Y -35.087,Z -65.276,A -90.000,B 90.000,C 0.000} C_DIS
LIN {X -13.328,Y -35.052,Z -65.014,A -90.000,B 90.000,C 0.000} C_DIS
LIN {X -13.099,Y -35.014,Z -64.767,A -90.000,B 90.000,C 0.000} C_DIS
LIN {X -12.967,Y -34.993,Z -64.634,A -90.000,B 90.000,C 0.000} C_DIS
LIN {X -12.848,Y -34.976,Z -64.519,A -90.000,B 90.000,C 0.000} C_DIS
LIN {X -12.715,Y -34.961,Z -64.410,A -90.000,B 90.000,C 0.000} C_DIS
LIN {X -12.604,Y -34.950,Z -64.331,A -90.000,B 90.000,C 0.000} C_DIS
LIN {X -12.462,Y -34.929,Z -64.248,A -90.000,B 90.000,C 0.000} C_DIS
LIN {X -12.314,Y -34.909,Z -64.169,A -90.000,B 90.000,C 0.000} C_DIS
LIN {X -12.124,Y -34.886,Z -64.079,A -90.000,B 90.000,C 0.000} C_DIS
LIN {X -11.951,Y -34.872,Z -64.017,A -90.000,B 90.000,C 0.000} C_DIS
LIN {X -11.857,Y -34.866,Z -63.990,A -90.000,B 90.000,C 0.000} C_DIS
LIN {X -10.965,Y -34.789,Z -63.762,A -90.000,B 90.000,C 0.000} C_DIS
LIN {X -10.857,Y -34.782,Z -63.738,A -90.000,B 90.000,C 0.000} C_DIS
LIN {X -10.426,Y -34.753,Z -63.648,A -90.000,B 90.000,C 0.000} C_DIS
LIN {X -10.294,Y -34.745,Z -63.625,A -90.000,B 90.000,C 0.000} C_DIS
LIN {X -9.487,Y -34.696,Z -63.512,A -90.000,B 90.000,C 0.000} C_DIS
LIN {X -9.071,Y -34.664,Z -63.457,A -90.000,B 90.000,C 0.000} C_DIS
LIN {X -8.722,Y -34.627,Z -63.415,A -90.000,B 90.000,C 0.000} C_DIS
LIN {X -8.660,Y -34.621,Z -63.409,A -90.000,B 90.000,C 0.000} C_DIS
LIN {X -8.491,Y -34.609,Z -63.402,A -90.000,B 90.000,C 0.000} C_DIS
LIN {X -6.653,Y -34.518,Z -63.391,A -90.000,B 90.000,C 0.000} C_DIS
LIN {X -6.559,Y -34.514,Z -63.393,A -90.000,B 90.000,C 0.000} C_DIS
LIN {X -5.894,Y -34.496,Z -63.417,A -90.000,B 90.000,C 0.000} C_DIS
LIN {X -5.183,Y -34.466,Z -63.432,A -90.000,B 90.000,C 0.000} C_DIS
LIN {X -3.985,Y -34.426,Z -63.453,A -90.000,B 90.000,C 0.000} C_DIS
LIN {X -3.742,Y -34.413,Z -63.461,A -90.000,B 90.000,C 0.000} C_DIS
LIN {X -1.930,Y -34.341,Z -63.556,A -90.000,B 90.000,C 0.000} C_DIS
LIN {X -1.469,Y -34.315,Z -63.569,A -90.000,B 90.000,C 0.000} C_DIS
LIN {X 0.056,Y -34.273,Z -63.590,A -90.000,B 90.000,C 0.000} C_DIS
LIN {X 1.106,Y -34.244,Z -63.607,A -90.000,B 90.000,C 0.000} C_DIS
LIN {X 1.562,Y -34.234,Z -63.618,A -90.000,B 90.000,C 0.000} C_DIS
LIN {X 1.651,Y -34.230,Z -63.617,A -90.000,B 90.000,C 0.000} C_DIS
LIN {X 1.885,Y -34.213,Z -63.620,A -90.000,B 90.000,C 0.000} C_DIS
LIN {X 2.404,Y -34.189,Z -63.620,A -90.000,B 90.000,C 0.000} C_DIS
LIN {X 3.086,Y -34.169,Z -63.633,A -90.000,B 90.000,C 0.000} C_DIS
LIN {X 4.439,Y -34.125,Z -63.665,A -90.000,B 90.000,C 0.000} C_DIS
LIN {X 4.629,Y -34.113,Z -63.663,A -90.000,B 90.000,C 0.000} C_DIS
LIN {X 5.918,Y -34.057,Z -63.639,A -90.000,B 90.000,C 0.000} C_DIS
LIN {X 6.812,Y -34.036,Z -63.643,A -90.000,B 90.000,C 0.000} C_DIS
LIN {X 7.253,Y -34.031,Z -63.645,A -90.000,B 90.000,C 0.000} C_DIS
LIN {X 7.580,Y -34.024,Z -63.652,A -90.000,B 90.000,C 0.000} C_DIS
LIN {X 8.566,Y -34.017,Z -63.687,A -90.000,B 90.000,C 0.000} C_DIS
LIN {X 8.811,Y -34.023,Z -63.690,A -90.000,B 90.000,C 0.000} C_DIS
LIN {X 9.227,Y -34.024,Z -63.700,A -90.000,B 90.000,C 0.000} C_DIS
LIN {X 9.654,Y -34.029,Z -63.720,A -90.000,B 90.000,C 0.000} C_DIS
LIN {X 9.979,Y -34.036,Z -63.739,A -90.000,B 90.000,C 0.000} C_DIS
LIN {X 10.295,Y -34.063,Z -63.742,A -90.000,B 90.000,C 0.000} C_DIS
LIN {X 10.530,Y -34.071,Z -63.754,A -90.000,B 90.000,C 0.000} C_DIS
LIN {X 10.786,Y -34.072,Z -63.758,A -90.000,B 90.000,C 0.000} C_DIS
LIN {X 10.996,Y -34.077,Z -63.765,A -90.000,B 90.000,C 0.000} C_DIS
LIN {X 11.243,Y -34.106,Z -63.758,A -90.000,B 90.000,C 0.000} C_DIS
LIN {X 11.398,Y -34.127,Z -63.757,A -90.000,B 90.000,C 0.000} C_DIS
LIN {X 11.555,Y -34.141,Z -63.763,A -90.000,B 90.000,C 0.000} C_DIS
LIN {X 11.677,Y -34.096,Z -63.695,A -90.000,B 90.000,C 0.000} C_DIS
LIN {X 11.964,Y -34.027,Z -63.507,A -90.000,B 90.000,C 0.000} C_DIS
LIN {X 12.243,Y -33.990,Z -63.293,A -90.000,B 90.000,C 0.000} C_DIS
LIN {X 12.311,Y -33.984,Z -63.238,A -90.000,B 90.000,C 0.000} C_DIS
LIN {X 12.490,Y -33.975,Z -63.087,A -90.000,B 90.000,C 0.000} C_DIS
LIN {X 12.555,Y -33.972,Z -63.039,A -90.000,B 90.000,C 0.000} C_DIS
LIN {X 12.822,Y -33.971,Z -62.854,A -90.000,B 90.000,C 0.000} C_DIS
LIN {X 12.998,Y -33.967,Z -62.739,A -90.000,B 90.000,C 0.000} C_DIS
LIN {X 13.095,Y -33.970,Z -62.681,A -90.000,B 90.000,C 0.000} C_DIS
LIN {X 13.445,Y -33.987,Z -62.484,A -90.000,B 90.000,C 0.000} C_DIS
LIN {X 13.799,Y -33.987,Z -62.301,A -90.000,B 90.000,C 0.000} C_DIS
LIN {X 14.065,Y -33.971,Z -62.184,A -90.000,B 90.000,C 0.000} C_DIS
LIN {X 14.189,Y -33.968,Z -62.136,A -90.000,B 90.000,C 0.000} C_DIS
LIN {X 14.598,Y -33.966,Z -61.993,A -90.000,B 90.000,C 0.000} C_DIS
LIN {X 14.743,Y -33.972,Z -61.949,A -90.000,B 90.000,C 0.000} C_DIS
LIN {X 14.820,Y -33.975,Z -61.928,A -90.000,B 90.000,C 0.000} C_DIS
LIN {X 15.169,Y -33.979,Z -61.851,A -90.000,B 90.000,C 0.000} C_DIS
LIN {X 15.212,Y -33.980,Z -61.843,A -90.000,B 90.000,C 0.000} C_DIS
LIN {X 15.569,Y -33.981,Z -61.806,A -90.000,B 90.000,C 0.000} C_DIS
LIN {X 15.613,Y -33.981,Z -61.802,A -90.000,B 90.000,C 0.000} C_DIS
LIN {X 16.199,Y -33.967,Z -61.765,A -90.000,B 90.000,C 0.000} C_DIS
LIN {X 16.420,Y -33.956,Z -61.758,A -90.000,B 90.000,C 0.000} C_DIS
LIN {X 16.595,Y -33.955,Z -61.761,A -90.000,B 90.000,C 0.000} C_DIS
LIN {X 16.677,Y -33.955,Z -61.763,A -90.000,B 90.000,C 0.000} C_DIS
LIN {X 16.924,Y -33.941,Z -61.782,A -90.000,B 90.000,C 0.000} C_DIS
LIN {X 17.077,Y -33.937,Z -61.798,A -90.000,B 90.000,C 0.000} C_DIS
LIN {X 17.692,Y -33.935,Z -61.882,A -90.000,B 90.000,C 0.000} C_DIS
LIN {X 17.771,Y -33.897,Z -61.860,A -90.000,B 90.000,C 0.000} C_DIS
LIN {X 17.874,Y -33.885,Z -61.793,A -90.000,B 90.000,C 0.000} C_DIS
LIN {X 17.947,Y -33.879,Z -61.748,A -90.000,B 90.000,C 0.000} C_DIS
LIN {X 18.111,Y -33.865,Z -61.652,A -90.000,B 90.000,C 0.000} C_DIS
LIN {X 18.320,Y -33.839,Z -61.543,A -90.000,B 90.000,C 0.000} C_DIS
LIN {X 18.446,Y -33.841,Z -61.454,A -90.000,B 90.000,C 0.000} C_DIS
LIN {X 18.520,Y -33.843,Z -61.403,A -90.000,B 90.000,C 0.000} C_DIS
LIN {X 18.713,Y -33.859,Z -61.282,A -90.000,B 90.000,C 0.000} C_DIS
LIN {X 18.968,Y -33.862,Z -61.148,A -90.000,B 90.000,C 0.000} C_DIS
LIN {X 19.086,Y -33.868,Z -61.090,A -90.000,B 90.000,C 0.000} C_DIS
LIN {X 19.499,Y -33.873,Z -60.933,A -90.000,B 90.000,C 0.000} C_DIS
LIN {X 19.618,Y -33.879,Z -60.891,A -90.000,B 90.000,C 0.000} C_DIS
LIN {X 20.028,Y -33.886,Z -60.789,A -90.000,B 90.000,C 0.000} C_DIS
LIN {X 20.141,Y -33.883,Z -60.771,A -90.000,B 90.000,C 0.000} C_DIS
LIN {X 20.447,Y -33.888,Z -60.732,A -90.000,B 90.000,C 0.000} C_DIS
LIN {X 20.624,Y -33.881,Z -60.721,A -90.000,B 90.000,C 0.000} C_DIS
LIN {X 20.785,Y -33.881,Z -60.717,A -90.000,B 90.000,C 0.000} C_DIS
LIN {X 20.870,Y -33.883,Z -60.717,A -90.000,B 90.000,C 0.000} C_DIS
LIN {X 21.167,Y -33.871,Z -60.735,A -90.000,B 90.000,C 0.000} C_DIS
LIN {X 21.291,Y -33.868,Z -60.743,A -90.000,B 90.000,C 0.000} C_DIS
LIN {X 21.379,Y -33.860,Z -60.754,A -90.000,B 90.000,C 0.000} C_DIS
LIN {X 21.438,Y -33.859,Z -60.760,A -90.000,B 90.000,C 0.000} C_DIS
LIN {X 21.851,Y -33.843,Z -60.835,A -90.000,B 90.000,C 0.000} C_DIS
LIN {X 21.994,Y -33.831,Z -60.874,A -90.000,B 90.000,C 0.000} C_DIS
LIN {X 22.188,Y -33.928,Z -60.814,A -90.000,B 90.000,C 0.000} C_DIS
LIN {X 22.249,Y -33.960,Z -60.798,A -90.000,B 90.000,C 0.000} C_DIS
LIN {X 22.481,Y -33.962,Z -60.627,A -90.000,B 90.000,C 0.000} C_DIS
LIN {X 22.691,Y -33.965,Z -60.475,A -90.000,B 90.000,C 0.000} C_DIS
LIN {X 22.922,Y -33.966,Z -60.314,A -90.000,B 90.000,C 0.000} C_DIS
LIN {X 23.232,Y -33.964,Z -60.106,A -90.000,B 90.000,C 0.000} C_DIS
LIN {X 23.513,Y -33.958,Z -59.932,A -90.000,B 90.000,C 0.000} C_DIS
LIN {X 23.744,Y -33.953,Z -59.795,A -90.000,B 90.000,C 0.000} C_DIS
LIN {X 24.088,Y -33.947,Z -59.603,A -90.000,B 90.000,C 0.000} C_DIS
LIN {X 24.182,Y -33.946,Z -59.551,A -90.000,B 90.000,C 0.000} C_DIS
LIN {X 24.474,Y -33.937,Z -59.402,A -90.000,B 90.000,C 0.000} C_DIS
LIN {X 24.925,Y -33.918,Z -59.189,A -90.000,B 90.000,C 0.000} C_DIS
LIN {X 24.961,Y -33.878,Z -59.140,A -90.000,B 90.000,C 0.000} C_DIS
LIN {X 25.075,Y -33.769,Z -59.017,A -90.000,B 90.000,C 0.000} C_DIS
LIN {X 25.164,Y -33.695,Z -58.928,A -90.000,B 90.000,C 0.000} C_DIS
LIN {X 25.179,Y -33.684,Z -58.914,A -90.000,B 90.000,C 0.000} C_DIS
LIN {X 25.269,Y -33.621,Z -58.838,A -90.000,B 90.000,C 0.000} C_DIS
LIN {X 25.328,Y -33.584,Z -58.791,A -90.000,B 90.000,C 0.000} C_DIS
LIN {X 25.394,Y -33.547,Z -58.742,A -90.000,B 90.000,C 0.000} C_DIS
LIN {X 25.506,Y -33.491,Z -58.664,A -90.000,B 90.000,C 0.000} C_DIS
LIN {X 25.629,Y -33.438,Z -58.584,A -90.000,B 90.000,C 0.000} C_DIS
LIN {X 25.700,Y -33.413,Z -58.543,A -90.000,B 90.000,C 0.000} C_DIS
LIN {X 25.768,Y -33.391,Z -58.507,A -90.000,B 90.000,C 0.000} C_DIS
LIN {X 25.740,Y -33.398,Z -58.265,A -90.000,B 90.000,C 0.000} C_DIS
LIN {X 25.729,Y -33.402,Z -58.134,A -90.000,B 90.000,C 0.000} C_DIS
LIN {X 25.716,Y -33.412,Z -57.965,A -90.000,B 90.000,C 0.000} C_DIS
LIN {X 25.695,Y -33.435,Z -57.513,A -90.000,B 90.000,C 0.000} C_DIS
LIN {X 25.699,Y -33.439,Z -57.422,A -90.000,B 90.000,C 0.000} C_DIS
LIN {X 25.724,Y -33.461,Z -57.035,A -90.000,B 90.000,C 0.000} C_DIS
LIN {X 25.787,Y -33.480,Z -56.640,A -90.000,B 90.000,C 0.000} C_DIS
LIN {X 25.884,Y -33.504,Z -56.206,A -90.000,B 90.000,C 0.000} C_DIS
LIN {X 25.935,Y -33.509,Z -56.051,A -90.000,B 90.000,C 0.000} C_DIS
LIN {X 26.031,Y -33.527,Z -55.771,A -90.000,B 90.000,C 0.000} C_DIS
LIN {X 26.146,Y -33.533,Z -55.516,A -90.000,B 90.000,C 0.000} C_DIS
LIN {X 26.223,Y -33.541,Z -55.349,A -90.000,B 90.000,C 0.000} C_DIS
LIN {X 26.469,Y -33.550,Z -54.928,A -90.000,B 90.000,C 0.000} C_DIS
LIN {X 26.543,Y -33.555,Z -54.806,A -90.000,B 90.000,C 0.000} C_DIS
LIN {X 26.659,Y -33.559,Z -54.635,A -90.000,B 90.000,C 0.000} C_DIS
LIN {X 26.712,Y -33.562,Z -54.564,A -90.000,B 90.000,C 0.000} C_DIS
LIN {X 26.952,Y -33.568,Z -54.266,A -90.000,B 90.000,C 0.000} C_DIS
LIN {X 27.015,Y -33.569,Z -54.199,A -90.000,B 90.000,C 0.000} C_DIS
LIN {X 27.277,Y -33.575,Z -53.939,A -90.000,B 90.000,C 0.000} C_DIS
LIN {X 27.324,Y -33.574,Z -53.897,A -90.000,B 90.000,C 0.000} C_DIS
LIN {X 27.410,Y -33.574,Z -53.827,A -90.000,B 90.000,C 0.000} C_DIS
LIN {X 27.633,Y -33.579,Z -53.650,A -90.000,B 90.000,C 0.000} C_DIS
LIN {X 27.681,Y -33.578,Z -53.615,A -90.000,B 90.000,C 0.000} C_DIS
LIN {X 27.762,Y -33.575,Z -53.561,A -90.000,B 90.000,C 0.000} C_DIS
LIN {X 27.857,Y -33.574,Z -53.500,A -90.000,B 90.000,C 0.000} C_DIS
LIN {X 28.015,Y -33.578,Z -53.401,A -90.000,B 90.000,C 0.000} C_DIS
LIN {X 28.088,Y -33.577,Z -53.360,A -90.000,B 90.000,C 0.000} C_DIS
LIN {X 28.293,Y -33.573,Z -53.252,A -90.000,B 90.000,C 0.000} C_DIS
LIN {X 28.540,Y -33.573,Z -53.130,A -90.000,B 90.000,C 0.000} C_DIS
LIN {X 28.640,Y -33.574,Z -53.082,A -90.000,B 90.000,C 0.000} C_DIS
LIN {X 28.949,Y -33.565,Z -52.965,A -90.000,B 90.000,C 0.000} C_DIS
LIN {X 29.066,Y -33.564,Z -52.923,A -90.000,B 90.000,C 0.000} C_DIS
LIN {X 29.389,Y -33.561,Z -52.831,A -90.000,B 90.000,C 0.000} C_DIS
LIN {X 29.435,Y -33.621,Z -52.711,A -90.000,B 90.000,C 0.000} C_DIS
LIN {X 29.480,Y -33.666,Z -52.626,A -90.000,B 90.000,C 0.000} C_DIS
LIN {X 29.541,Y -33.684,Z -52.285,A -90.000,B 90.000,C 0.000} C_DIS
LIN {X 29.600,Y -33.688,Z -52.047,A -90.000,B 90.000,C 0.000} C_DIS
LIN {X 29.664,Y -33.695,Z -51.799,A -90.000,B 90.000,C 0.000} C_DIS
LIN {X 29.767,Y -33.710,Z -51.444,A -90.000,B 90.000,C 0.000} C_DIS
LIN {X 29.825,Y -33.719,Z -51.259,A -90.000,B 90.000,C 0.000} C_DIS
LIN {X 29.912,Y -33.719,Z -51.032,A -90.000,B 90.000,C 0.000} C_DIS
LIN {X 29.963,Y -33.723,Z -50.906,A -90.000,B 90.000,C 0.000} C_DIS
LIN {X 29.983,Y -33.726,Z -50.859,A -90.000,B 90.000,C 0.000} C_DIS
LIN {X 30.173,Y -33.735,Z -50.470,A -90.000,B 90.000,C 0.000} C_DIS
LIN {X 30.278,Y -33.741,Z -50.264,A -90.000,B 90.000,C 0.000} C_DIS
LIN {X 30.398,Y -33.744,Z -50.042,A -90.000,B 90.000,C 0.000} C_DIS
LIN {X 30.483,Y -33.747,Z -49.886,A -90.000,B 90.000,C 0.000} C_DIS
LIN {X 30.574,Y -33.742,Z -49.745,A -90.000,B 90.000,C 0.000} C_DIS
LIN {X 30.720,Y -33.742,Z -49.533,A -90.000,B 90.000,C 0.000} C_DIS
LIN {X 30.822,Y -33.739,Z -49.393,A -90.000,B 90.000,C 0.000} C_DIS
LIN {X 30.911,Y -33.740,Z -49.276,A -90.000,B 90.000,C 0.000} C_DIS
LIN {X 31.129,Y -33.754,Z -49.002,A -90.000,B 90.000,C 0.000} C_DIS
LIN {X 31.411,Y -33.756,Z -48.681,A -90.000,B 90.000,C 0.000} C_DIS
LIN {X 31.644,Y -33.740,Z -48.450,A -90.000,B 90.000,C 0.000} C_DIS
LIN {X 31.733,Y -33.737,Z -48.364,A -90.000,B 90.000,C 0.000} C_DIS
LIN {X 31.878,Y -33.729,Z -48.249,A -90.000,B 90.000,C 0.000} C_DIS
LIN {X 32.073,Y -33.721,Z -48.087,A -90.000,B 90.000,C 0.000} C_DIS
LIN {X 32.183,Y -33.720,Z -48.000,A -90.000,B 90.000,C 0.000} C_DIS
LIN {X 32.309,Y -33.723,Z -47.906,A -90.000,B 90.000,C 0.000} C_DIS
LIN {X 32.655,Y -33.727,Z -47.660,A -90.000,B 90.000,C 0.000} C_DIS
LIN {X 33.027,Y -33.716,Z -47.434,A -90.000,B 90.000,C 0.000} C_DIS
LIN {X 33.236,Y -33.697,Z -47.329,A -90.000,B 90.000,C 0.000} C_DIS
LIN {X 33.410,Y -33.689,Z -47.246,A -90.000,B 90.000,C 0.000} C_DIS
LIN {X 33.577,Y -33.674,Z -47.180,A -90.000,B 90.000,C 0.000} C_DIS
LIN {X 33.718,Y -33.665,Z -47.119,A -90.000,B 90.000,C 0.000} C_DIS
LIN {X 34.147,Y -33.663,Z -46.948,A -90.000,B 90.000,C 0.000} C_DIS
LIN {X 34.229,Y -33.661,Z -46.919,A -90.000,B 90.000,C 0.000} C_DIS
LIN {X 34.398,Y -33.659,Z -46.866,A -90.000,B 90.000,C 0.000} C_DIS
LIN {X 34.616,Y -33.659,Z -46.799,A -90.000,B 90.000,C 0.000} C_DIS
LIN {X 34.800,Y -33.654,Z -46.751,A -90.000,B 90.000,C 0.000} C_DIS
LIN {X 34.949,Y -33.654,Z -46.714,A -90.000,B 90.000,C 0.000} C_DIS
LIN {X 35.092,Y -33.651,Z -46.677,A -90.000,B 90.000,C 0.000} C_DIS
LIN {X 35.517,Y -33.619,Z -46.604,A -90.000,B 90.000,C 0.000} C_DIS
LIN {X 35.594,Y -33.611,Z -46.594,A -90.000,B 90.000,C 0.000} C_DIS
LIN {X 35.702,Y -33.604,Z -46.581,A -90.000,B 90.000,C 0.000} C_DIS
LIN {X 36.137,Y -33.583,Z -46.535,A -90.000,B 90.000,C 0.000} C_DIS
LIN {X 36.302,Y -33.583,Z -46.516,A -90.000,B 90.000,C 0.000} C_DIS
LIN {X 36.537,Y -33.587,Z -46.492,A -90.000,B 90.000,C 0.000} C_DIS
LIN {X 36.745,Y -33.585,Z -46.481,A -90.000,B 90.000,C 0.000} C_DIS
LIN {X 37.072,Y -33.590,Z -46.466,A -90.000,B 90.000,C 0.000} C_DIS
LIN {X 37.330,Y -33.586,Z -46.469,A -90.000,B 90.000,C 0.000} C_DIS
LIN {X 37.531,Y -33.581,Z -46.471,A -90.000,B 90.000,C 0.000} C_DIS
LIN {X 37.774,Y -33.565,Z -46.491,A -90.000,B 90.000,C 0.000} C_DIS
LIN {X 38.272,Y -33.535,Z -46.542,A -90.000,B 90.000,C 0.000} C_DIS
LIN {X 38.417,Y -33.526,Z -46.562,A -90.000,B 90.000,C 0.000} C_DIS
LIN {X 38.889,Y -33.511,Z -46.634,A -90.000,B 90.000,C 0.000} C_DIS
LIN {X 39.244,Y -33.509,Z -46.693,A -90.000,B 90.000,C 0.000} C_DIS
LIN {X 39.615,Y -33.502,Z -46.772,A -90.000,B 90.000,C 0.000} C_DIS
LIN {X 40.380,Y -33.492,Z -46.935,A -90.000,B 90.000,C 0.000} C_DIS
LIN {X 40.713,Y -33.490,Z -47.007,A -90.000,B 90.000,C 0.000} C_DIS
LIN {X 40.973,Y -33.498,Z -47.056,A -90.000,B 90.000,C 0.000} C_DIS
LIN {X 41.699,Y -33.530,Z -47.200,A -90.000,B 90.000,C 0.000} C_DIS
LIN {X 42.233,Y -33.582,Z -47.259,A -90.000,B 90.000,C 0.000} C_DIS
LIN {X 42.389,Y -33.595,Z -47.274,A -90.000,B 90.000,C 0.000} C_DIS
LIN {X 42.655,Y -33.641,Z -47.264,A -90.000,B 90.000,C 0.000} C_DIS
LIN {X 43.033,Y -33.712,Z -47.254,A -90.000,B 90.000,C 0.000} C_DIS
LIN {X 43.363,Y -33.756,Z -47.232,A -90.000,B 90.000,C 0.000} C_DIS
LIN {X 43.459,Y -33.773,Z -47.222,A -90.000,B 90.000,C 0.000} C_DIS
LIN {X 44.023,Y -33.804,Z -47.107,A -90.000,B 90.000,C 0.000} C_DIS
LIN {X 44.437,Y -33.814,Z -47.011,A -90.000,B 90.000,C 0.000} C_DIS
LIN {X 44.727,Y -33.822,Z -46.941,A -90.000,B 90.000,C 0.000} C_DIS
LIN {X 44.854,Y -33.825,Z -46.910,A -90.000,B 90.000,C 0.000} C_DIS
LIN {X 45.534,Y -33.813,Z -46.773,A -90.000,B 90.000,C 0.000} C_DIS
LIN {X 45.662,Y -33.814,Z -46.749,A -90.000,B 90.000,C 0.000} C_DIS
LIN {X 46.093,Y -33.824,Z -46.677,A -90.000,B 90.000,C 0.000} C_DIS
LIN {X 46.619,Y -33.845,Z -46.595,A -90.000,B 90.000,C 0.000} C_DIS
LIN {X 46.690,Y -33.850,Z -46.582,A -90.000,B 90.000,C 0.000} C_DIS
LIN {X 47.133,Y -33.856,Z -46.524,A -90.000,B 90.000,C 0.000} C_DIS
LIN {X 47.199,Y -33.854,Z -46.517,A -90.000,B 90.000,C 0.000} C_DIS
LIN {X 47.546,Y -33.831,Z -46.491,A -90.000,B 90.000,C 0.000} C_DIS
LIN {X 47.780,Y -33.811,Z -46.480,A -90.000,B 90.000,C 0.000} C_DIS
LIN {X 47.918,Y -33.796,Z -46.478,A -90.000,B 90.000,C 0.000} C_DIS
LIN {X 48.060,Y -33.786,Z -46.480,A -90.000,B 90.000,C 0.000} C_DIS
LIN {X 48.468,Y -33.767,Z -46.494,A -90.000,B 90.000,C 0.000} C_DIS
LIN {X 48.547,Y -33.764,Z -46.498,A -90.000,B 90.000,C 0.000} C_DIS
LIN {X 49.062,Y -33.768,Z -46.540,A -90.000,B 90.000,C 0.000} C_DIS
LIN {X 49.730,Y -33.779,Z -46.603,A -90.000,B 90.000,C 0.000} C_DIS
LIN {X 50.051,Y -33.782,Z -46.636,A -90.000,B 90.000,C 0.000} C_DIS
LIN {X 50.659,Y -33.764,Z -46.727,A -90.000,B 90.000,C 0.000} C_DIS
LIN {X 51.053,Y -33.731,Z -46.812,A -90.000,B 90.000,C 0.000} C_DIS
LIN {X 51.625,Y -33.669,Z -46.955,A -90.000,B 90.000,C 0.000} C_DIS
LIN {X 51.953,Y -33.641,Z -47.051,A -90.000,B 90.000,C 0.000} C_DIS
LIN {X 52.279,Y -33.621,Z -47.151,A -90.000,B 90.000,C 0.000} C_DIS
LIN {X 52.526,Y -33.606,Z -47.247,A -90.000,B 90.000,C 0.000} C_DIS
LIN {X 52.837,Y -33.597,Z -47.372,A -90.000,B 90.000,C 0.000} C_DIS
LIN {X 52.975,Y -33.596,Z -47.430,A -90.000,B 90.000,C 0.000} C_DIS
LIN {X 53.192,Y -33.599,Z -47.526,A -90.000,B 90.000,C 0.000} C_DIS
LIN {X 53.388,Y -33.605,Z -47.616,A -90.000,B 90.000,C 0.000} C_DIS
LIN {X 53.504,Y -33.609,Z -47.670,A -90.000,B 90.000,C 0.000} C_DIS
LIN {X 53.893,Y -33.618,Z -47.903,A -90.000,B 90.000,C 0.000} C_DIS
LIN {X 55.371,Y -33.604,Z -48.875,A -90.000,B 90.000,C 0.000} C_DIS
LIN {X 56.644,Y -33.602,Z -49.726,A -90.000,B 90.000,C 0.000} C_DIS
LIN {X 56.889,Y -33.598,Z -49.905,A -90.000,B 90.000,C 0.000} C_DIS
LIN {X 57.028,Y -33.597,Z -50.008,A -90.000,B 90.000,C 0.000} C_DIS
LIN {X 59.394,Y -33.598,Z -52.020,A -90.000,B 90.000,C 0.000} C_DIS
LIN {X 59.743,Y -33.592,Z -52.339,A -90.000,B 90.000,C 0.000} C_DIS
LIN {X 60.327,Y -33.592,Z -52.892,A -90.000,B 90.000,C 0.000} C_DIS
LIN {X 60.956,Y -33.594,Z -53.489,A -90.000,B 90.000,C 0.000} C_DIS
LIN {X 62.048,Y -33.606,Z -54.535,A -90.000,B 90.000,C 0.000} C_DIS
LIN {X 63.175,Y -33.635,Z -55.649,A -90.000,B 90.000,C 0.000} C_DIS
LIN {X 63.380,Y -33.639,Z -55.854,A -90.000,B 90.000,C 0.000} C_DIS
LIN {X 64.134,Y -33.665,Z -56.616,A -90.000,B 90.000,C 0.000} C_DIS
LIN {X 64.474,Y -33.682,Z -56.948,A -90.000,B 90.000,C 0.000} C_DIS
LIN {X 65.781,Y -33.760,Z -58.236,A -90.000,B 90.000,C 0.000} C_DIS
LIN {X 66.084,Y -33.780,Z -58.532,A -90.000,B 90.000,C 0.000} C_DIS
LIN {X 66.729,Y -33.819,Z -59.170,A -90.000,B 90.000,C 0.000} C_DIS
LIN {X 67.515,Y -33.852,Z -60.008,A -90.000,B 90.000,C 0.000} C_DIS
LIN {X 67.773,Y -33.863,Z -60.289,A -90.000,B 90.000,C 0.000} C_DIS
LIN {X 68.123,Y -33.869,Z -60.689,A -90.000,B 90.000,C 0.000} C_DIS
LIN {X 68.381,Y -33.874,Z -60.998,A -90.000,B 90.000,C 0.000} C_DIS
LIN {X 69.982,Y -33.961,Z -63.014,A -90.000,B 90.000,C 0.000} C_DIS
LIN {X 70.772,Y -33.986,Z -64.043,A -90.000,B 90.000,C 0.000} C_DIS
LIN {X 71.600,Y -33.987,Z -65.165,A -90.000,B 90.000,C 0.000} C_DIS
LIN {X 72.085,Y -33.973,Z -65.846,A -90.000,B 90.000,C 0.000} C_DIS
LIN {X 72.271,Y -33.981,Z -66.089,A -90.000,B 90.000,C 0.000} C_DIS
LIN {X 72.418,Y -33.977,Z -66.265,A -90.000,B 90.000,C 0.000} C_DIS
LIN {X 72.930,Y -33.971,Z -66.892,A -90.000,B 90.000,C 0.000} C_DIS
LIN {X 73.059,Y -33.964,Z -67.057,A -90.000,B 90.000,C 0.000} C_DIS
LIN {X 73.164,Y -33.953,Z -67.179,A -90.000,B 90.000,C 0.000} C_DIS
LIN {X 73.236,Y -33.947,Z -67.267,A -90.000,B 90.000,C 0.000} C_DIS
LIN {X 73.590,Y -33.930,Z -67.720,A -90.000,B 90.000,C 0.000} C_DIS
LIN {X 73.686,Y -33.933,Z -67.831,A -90.000,B 90.000,C 0.000} C_DIS
LIN {X 73.871,Y -33.925,Z -68.021,A -90.000,B 90.000,C 0.000} C_DIS
LIN {X 73.999,Y -33.917,Z -68.157,A -90.000,B 90.000,C 0.000} C_DIS
LIN {X 74.062,Y -33.913,Z -68.224,A -90.000,B 90.000,C 0.000} C_DIS
LIN {X 74.234,Y -33.893,Z -68.419,A -90.000,B 90.000,C 0.000} C_DIS
LIN {X 74.330,Y -33.889,Z -68.517,A -90.000,B 90.000,C 0.000} C_DIS
LIN {X 74.434,Y -33.890,Z -68.629,A -90.000,B 90.000,C 0.000} C_DIS
LIN {X 74.467,Y -33.891,Z -68.666,A -90.000,B 90.000,C 0.000} C_DIS
LIN {X 74.606,Y -33.886,Z -68.809,A -90.000,B 90.000,C 0.000} C_DIS
LIN {X 74.973,Y -33.866,Z -69.199,A -90.000,B 90.000,C 0.000} C_DIS
LIN {X 75.163,Y -33.862,Z -69.393,A -90.000,B 90.000,C 0.000} C_DIS
LIN {X 75.690,Y -33.826,Z -69.970,A -90.000,B 90.000,C 0.000} C_DIS
LIN {X 75.936,Y -33.826,Z -70.216,A -90.000,B 90.000,C 0.000} C_DIS
LIN {X 76.194,Y -33.822,Z -70.479,A -90.000,B 90.000,C 0.000} C_DIS
LIN {X 76.435,Y -33.806,Z -70.749,A -90.000,B 90.000,C 0.000} C_DIS
LIN {X 76.656,Y -33.800,Z -70.988,A -90.000,B 90.000,C 0.000} C_DIS
LIN {X 76.956,Y -33.800,Z -71.319,A -90.000,B 90.000,C 0.000} C_DIS
LIN {X 77.177,Y -33.625,Z -71.362,A -90.000,B 90.000,C 0.000} C_DIS
LIN {X 77.199,Y -33.613,Z -71.372,A -90.000,B 90.000,C 0.000} C_DIS
LIN {X 77.252,Y -33.579,Z -71.392,A -90.000,B 90.000,C 0.000} C_DIS
LIN {X 77.317,Y -33.540,Z -71.418,A -90.000,B 90.000,C 0.000} C_DIS
LIN {X 77.483,Y -33.453,Z -71.501,A -90.000,B 90.000,C 0.000} C_DIS
LIN {X 77.564,Y -33.418,Z -71.555,A -90.000,B 90.000,C 0.000} C_DIS
LIN {X 77.658,Y -33.383,Z -71.625,A -90.000,B 90.000,C 0.000} C_DIS
LIN {X 77.754,Y -33.354,Z -71.705,A -90.000,B 90.000,C 0.000} C_DIS
LIN {X 77.867,Y -33.330,Z -71.809,A -90.000,B 90.000,C 0.000} C_DIS
LIN {X 78.015,Y -33.311,Z -71.962,A -90.000,B 90.000,C 0.000} C_DIS
LIN {X 78.092,Y -33.308,Z -72.049,A -90.000,B 90.000,C 0.000} C_DIS
LIN {X 78.114,Y -33.308,Z -71.969,A -90.000,B 90.000,C 0.000} C_DIS
LIN {X 78.106,Y -33.308,Z -71.949,A -90.000,B 90.000,C 0.000} C_DIS
LIN {X 78.123,Y -33.308,Z -71.941,A -90.000,B 90.000,C 0.000} C_DIS
LIN {X 78.203,Y -33.311,Z -71.696,A -90.000,B 90.000,C 0.000} C_DIS
LIN {X 78.266,Y -33.308,Z -71.506,A -90.000,B 90.000,C 0.000} C_DIS
LIN {X 78.412,Y -33.293,Z -71.031,A -90.000,B 90.000,C 0.000} C_DIS
LIN {X 78.575,Y -33.308,Z -70.563,A -90.000,B 90.000,C 0.000} C_DIS
LIN {X 78.603,Y -33.310,Z -70.478,A -90.000,B 90.000,C 0.000} C_DIS
LIN {X 78.624,Y -33.308,Z -70.415,A -90.000,B 90.000,C 0.000} C_DIS
LIN {X 78.681,Y -36.449,Z -70.240,A -90.000,B 90.000,C 0.000} C_DIS
LIN {X 78.689,Y -36.457,Z -70.218,A -90.000,B 90.000,C 0.000} C_DIS
LIN {X 78.689,Y -36.460,Z -70.216,A -90.000,B 90.000,C 0.000} C_DIS
LIN {X 78.691,Y -36.502,Z -70.212,A -90.000,B 90.000,C 0.000} C_DIS
LIN {X 78.699,Y -36.543,Z -70.190,A -90.000,B 90.000,C 0.000} C_DIS
LIN {X 78.758,Y -33.308,Z -70.015,A -90.000,B 90.000,C 0.000} C_DIS
LIN {X 78.776,Y -33.308,Z -69.961,A -90.000,B 90.000,C 0.000} C_DIS
LIN {X 78.776,Y -60.000,Z -69.961,A -90.000,B 90.000,C 0.000} C_DIS
LIN {X 89.535,Y -60.000,Z -54.092,A -90.000,B 90.000,C 0.000} C_DIS
LIN {X 89.535,Y -33.308,Z -54.092,A -90.000,B 90.000,C 0.000} C_DIS
LIN {X 89.682,Y -33.308,Z -53.958,A -90.000,B 90.000,C 0.000} C_DIS
LIN {X 89.861,Y -33.308,Z -53.777,A -90.000,B 90.000,C 0.000} C_DIS
LIN {X 89.990,Y -33.306,Z -53.654,A -90.000,B 90.000,C 0.000} C_DIS
LIN {X 90.003,Y -33.307,Z -53.657,A -90.000,B 90.000,C 0.000} C_DIS
LIN {X 90.338,Y -33.308,Z -53.373,A -90.000,B 90.000,C 0.000} C_DIS
LIN {X 90.695,Y -33.310,Z -53.067,A -90.000,B 90.000,C 0.000} C_DIS
LIN {X 90.715,Y -33.308,Z -53.050,A -90.000,B 90.000,C 0.000} C_DIS
LIN {X 90.809,Y -46.534,Z -52.971,A -90.000,B 90.000,C 0.000} C_DIS
LIN {X 90.902,Y -46.602,Z -52.894,A -90.000,B 90.000,C 0.000} C_DIS
LIN {X 90.994,Y -46.683,Z -52.821,A -90.000,B 90.000,C 0.000} C_DIS
LIN {X 91.177,Y -46.853,Z -52.683,A -90.000,B 90.000,C 0.000} C_DIS
LIN {X 91.357,Y -47.025,Z -52.556,A -90.000,B 90.000,C 0.000} C_DIS
LIN {X 91.623,Y -47.279,Z -52.386,A -90.000,B 90.000,C 0.000} C_DIS
LIN {X 91.796,Y -47.445,Z -52.285,A -90.000,B 90.000,C 0.000} C_DIS
LIN {X 91.967,Y -47.606,Z -52.193,A -90.000,B 90.000,C 0.000} C_DIS
LIN {X 92.134,Y -47.764,Z -52.111,A -90.000,B 90.000,C 0.000} C_DIS
LIN {X 92.299,Y -47.918,Z -52.037,A -90.000,B 90.000,C 0.000} C_DIS
LIN {X 92.460,Y -48.065,Z -51.972,A -90.000,B 90.000,C 0.000} C_DIS
LIN {X 92.619,Y -48.199,Z -51.915,A -90.000,B 90.000,C 0.000} C_DIS
LIN {X 92.696,Y -48.267,Z -51.889,A -90.000,B 90.000,C 0.000} C_DIS
LIN {X 92.850,Y -48.409,Z -51.843,A -90.000,B 90.000,C 0.000} C_DIS
LIN {X 93.000,Y -48.547,Z -51.803,A -90.000,B 90.000,C 0.000} C_DIS
LIN {X 93.147,Y -48.679,Z -51.771,A -90.000,B 90.000,C 0.000} C_DIS
LIN {X 93.290,Y -48.804,Z -51.744,A -90.000,B 90.000,C 0.000} C_DIS
LIN {X 93.430,Y -48.923,Z -51.724,A -90.000,B 90.000,C 0.000} C_DIS
LIN {X 93.566,Y -49.036,Z -51.708,A -90.000,B 90.000,C 0.000} C_DIS
LIN {X 93.699,Y -49.144,Z -51.698,A -90.000,B 90.000,C 0.000} C_DIS
LIN {X 93.891,Y -49.295,Z -51.690,A -90.000,B 90.000,C 0.000} C_DIS
LIN {X 94.014,Y -49.390,Z -51.690,A -90.000,B 90.000,C 0.000} C_DIS
LIN {X 94.249,Y -49.565,Z -51.700,A -90.000,B 90.000,C 0.000} C_DIS
LIN {X 94.468,Y -49.720,Z -51.721,A -90.000,B 90.000,C 0.000} C_DIS
LIN {X 94.571,Y -49.790,Z -51.734,A -90.000,B 90.000,C 0.000} C_DIS
LIN {X 94.764,Y -49.918,Z -51.765,A -90.000,B 90.000,C 0.000} C_DIS
LIN {X 94.940,Y -50.027,Z -51.798,A -90.000,B 90.000,C 0.000} C_DIS
LIN {X 95.098,Y -50.120,Z -51.831,A -90.000,B 90.000,C 0.000} C_DIS
LIN {X 95.238,Y -50.195,Z -51.860,A -90.000,B 90.000,C 0.000} C_DIS
LIN {X 95.358,Y -50.254,Z -51.881,A -90.000,B 90.000,C 0.000} C_DIS
LIN {X 95.459,Y -50.297,Z -51.892,A -90.000,B 90.000,C 0.000} C_DIS
LIN {X 95.502,Y -50.312,Z -51.893,A -90.000,B 90.000,C 0.000} C_DIS
LIN {X 95.540,Y -50.323,Z -51.890,A -90.000,B 90.000,C 0.000} C_DIS
LIN {X 95.573,Y -50.329,Z -51.883,A -90.000,B 90.000,C 0.000} C_DIS
LIN {X 95.600,Y -50.331,Z -51.871,A -90.000,B 90.000,C 0.000} C_DIS
LIN {X 95.623,Y -50.329,Z -51.854,A -90.000,B 90.000,C 0.000} C_DIS
LIN {X 95.632,Y -50.326,Z -51.843,A -90.000,B 90.000,C 0.000} C_DIS
LIN {X 95.646,Y -50.315,Z -51.818,A -90.000,B 90.000,C 0.000} C_DIS
LIN {X 95.651,Y -50.308,Z -51.803,A -90.000,B 90.000,C 0.000} C_DIS
LIN {X 95.658,Y -50.278,Z -51.749,A -90.000,B 90.000,C 0.000} C_DIS
LIN {X 95.652,Y -50.234,Z -51.679,A -90.000,B 90.000,C 0.000} C_DIS
LIN {X 95.641,Y -50.195,Z -51.623,A -90.000,B 90.000,C 0.000} C_DIS
LIN {X 95.624,Y -50.148,Z -51.560,A -90.000,B 90.000,C 0.000} C_DIS
LIN {X 95.601,Y -50.092,Z -51.488,A -90.000,B 90.000,C 0.000} C_DIS
LIN {X 95.538,Y -49.946,Z -51.317,A -90.000,B 90.000,C 0.000} C_DIS
LIN {X 95.498,Y -49.853,Z -51.218,A -90.000,B 90.000,C 0.000} C_DIS
LIN {X 95.451,Y -49.744,Z -51.109,A -90.000,B 90.000,C 0.000} C_DIS
LIN {X 95.398,Y -49.615,Z -50.990,A -90.000,B 90.000,C 0.000} C_DIS
LIN {X 95.339,Y -49.462,Z -50.859,A -90.000,B 90.000,C 0.000} C_DIS
LIN {X 95.274,Y -49.281,Z -50.718,A -90.000,B 90.000,C 0.000} C_DIS
LIN {X 95.124,Y -48.791,Z -50.401,A -90.000,B 90.000,C 0.000} C_DIS
LIN {X 95.039,Y -48.446,Z -50.224,A -90.000,B 90.000,C 0.000} C_DIS
LIN {X 94.948,Y -47.989,Z -50.034,A -90.000,B 90.000,C 0.000} C_DIS
LIN {X 94.850,Y -47.402,Z -49.831,A -90.000,B 90.000,C 0.000} C_DIS
LIN {X 94.798,Y -46.975,Z -49.724,A -90.000,B 90.000,C 0.000} C_DIS
LIN {X 94.772,Y -46.667,Z -49.669,A -90.000,B 90.000,C 0.000} C_DIS
LIN {X 94.759,Y -46.450,Z -49.642,A -90.000,B 90.000,C 0.000} C_DIS
LIN {X 94.752,Y -46.301,Z -49.628,A -90.000,B 90.000,C 0.000} C_DIS
LIN {X 94.745,Y -46.065,Z -49.614,A -90.000,B 90.000,C 0.000} C_DIS
LIN {X 94.745,Y -33.308,Z -49.614,A -90.000,B 90.000,C 0.000} C_DIS
LIN {X 94.733,Y -33.309,Z -49.588,A -90.000,B 90.000,C 0.000} C_DIS
LIN {X 94.686,Y -33.317,Z -49.425,A -90.000,B 90.000,C 0.000} C_DIS
LIN {X 94.652,Y -33.344,Z -49.197,A -90.000,B 90.000,C 0.000} C_DIS
LIN {X 94.656,Y -33.377,Z -49.002,A -90.000,B 90.000,C 0.000} C_DIS
LIN {X 94.669,Y -33.398,Z -48.893,A -90.000,B 90.000,C 0.000} C_DIS
LIN {X 94.685,Y -33.417,Z -48.802,A -90.000,B 90.000,C 0.000} C_DIS
LIN {X 94.706,Y -33.439,Z -48.703,A -90.000,B 90.000,C 0.000} C_DIS
LIN {X 94.734,Y -33.463,Z -48.599,A -90.000,B 90.000,C 0.000} C_DIS
LIN {X 94.877,Y -33.565,Z -48.195,A -90.000,B 90.000,C 0.000} C_DIS
LIN {X 94.922,Y -33.594,Z -48.090,A -90.000,B 90.000,C 0.000} C_DIS
LIN {X 95.199,Y -33.742,Z -47.563,A -90.000,B 90.000,C 0.000} C_DIS
LIN {X 95.304,Y -33.794,Z -47.377,A -90.000,B 90.000,C 0.000} C_DIS
LIN {X 95.630,Y -33.977,Z -46.799,A -90.000,B 90.000,C 0.000} C_DIS
LIN {X 95.743,Y -34.035,Z -46.621,A -90.000,B 90.000,C 0.000} C_DIS
LIN {X 95.879,Y -34.104,Z -46.414,A -90.000,B 90.000,C 0.000} C_DIS
LIN {X 96.153,Y -34.240,Z -46.016,A -90.000,B 90.000,C 0.000} C_DIS
LIN {X 96.221,Y -34.273,Z -45.922,A -90.000,B 90.000,C 0.000} C_DIS
LIN {X 96.341,Y -34.343,Z -45.749,A -90.000,B 90.000,C 0.000} C_DIS
LIN {X 96.409,Y -34.378,Z -45.654,A -90.000,B 90.000,C 0.000} C_DIS
LIN {X 96.525,Y -34.439,Z -45.488,A -90.000,B 90.000,C 0.000} C_DIS
LIN {X 96.511,Y -34.435,Z -45.404,A -90.000,B 90.000,C 0.000} C_DIS
LIN {X 96.503,Y -34.433,Z -45.323,A -90.000,B 90.000,C 0.000} C_DIS
LIN {X 96.487,Y -34.411,Z -45.032,A -90.000,B 90.000,C 0.000} C_DIS
LIN {X 96.477,Y -34.399,Z -44.919,A -90.000,B 90.000,C 0.000} C_DIS
LIN {X 96.470,Y -34.386,Z -44.785,A -90.000,B 90.000,C 0.000} C_DIS
LIN {X 96.469,Y -34.384,Z -44.753,A -90.000,B 90.000,C 0.000} C_DIS
LIN {X 96.470,Y -34.345,Z -44.456,A -90.000,B 90.000,C 0.000} C_DIS
LIN {X 96.485,Y -34.315,Z -44.286,A -90.000,B 90.000,C 0.000} C_DIS
LIN {X 96.512,Y -34.274,Z -44.038,A -90.000,B 90.000,C 0.000} C_DIS
LIN {X 96.532,Y -34.257,Z -43.914,A -90.000,B 90.000,C 0.000} C_DIS
LIN {X 96.589,Y -34.205,Z -43.627,A -90.000,B 90.000,C 0.000} C_DIS
LIN {X 96.613,Y -34.185,Z -43.534,A -90.000,B 90.000,C 0.000} C_DIS
LIN {X 96.658,Y -34.160,Z -43.392,A -90.000,B 90.000,C 0.000} C_DIS
LIN {X 96.712,Y -34.136,Z -43.232,A -90.000,B 90.000,C 0.000} C_DIS
LIN {X 96.783,Y -34.104,Z -43.030,A -90.000,B 90.000,C 0.000} C_DIS
LIN {X 96.851,Y -34.084,Z -42.860,A -90.000,B 90.000,C 0.000} C_DIS
LIN {X 96.890,Y -34.075,Z -42.768,A -90.000,B 90.000,C 0.000} C_DIS
LIN {X 97.031,Y -34.024,Z -42.471,A -90.000,B 90.000,C 0.000} C_DIS
LIN {X 97.089,Y -34.003,Z -42.355,A -90.000,B 90.000,C 0.000} C_DIS
LIN {X 97.185,Y -33.977,Z -42.179,A -90.000,B 90.000,C 0.000} C_DIS
LIN {X 97.292,Y -33.956,Z -41.996,A -90.000,B 90.000,C 0.000} C_DIS
LIN {X 97.386,Y -33.929,Z -41.855,A -90.000,B 90.000,C 0.000} C_DIS
LIN {X 97.765,Y -33.843,Z -41.316,A -90.000,B 90.000,C 0.000} C_DIS
LIN {X 97.801,Y -33.836,Z -41.266,A -90.000,B 90.000,C 0.000} C_DIS
LIN {X 97.873,Y -33.821,Z -41.183,A -90.000,B 90.000,C 0.000} C_DIS
LIN {X 98.246,Y -33.760,Z -40.763,A -90.000,B 90.000,C 0.000} C_DIS
LIN {X 98.427,Y -33.730,Z -40.565,A -90.000,B 90.000,C 0.000} C_DIS
LIN {X 98.775,Y -33.665,Z -40.233,A -90.000,B 90.000,C 0.000} C_DIS
LIN {X 98.950,Y -33.641,Z -40.071,A -90.000,B 90.000,C 0.000} C_DIS
LIN {X 99.073,Y -33.628,Z -39.961,A -90.000,B 90.000,C 0.000} C_DIS
LIN {X 99.348,Y -33.591,Z -39.741,A -90.000,B 90.000,C 0.000} C_DIS
LIN {X 99.809,Y -33.542,Z -39.381,A -90.000,B 90.000,C 0.000} C_DIS
LIN {X 99.939,Y -33.527,Z -39.290,A -90.000,B 90.000,C 0.000} C_DIS
LIN {X 100.173,Y -33.505,Z -39.130,A -90.000,B 90.000,C 0.000} C_DIS
LIN {X 100.707,Y -33.453,Z -38.790,A -90.000,B 90.000,C 0.000} C_DIS
LIN {X 100.951,Y -33.438,Z -38.637,A -90.000,B 90.000,C 0.000} C_DIS
LIN {X 101.649,Y -33.392,Z -38.249,A -90.000,B 90.000,C 0.000} C_DIS
LIN {X 101.826,Y -33.381,Z -38.155,A -90.000,B 90.000,C 0.000} C_DIS
LIN {X 102.282,Y -33.359,Z -37.937,A -90.000,B 90.000,C 0.000} C_DIS
LIN {X 102.819,Y -33.340,Z -37.681,A -90.000,B 90.000,C 0.000} C_DIS
LIN {X 103.319,Y -33.327,Z -37.454,A -90.000,B 90.000,C 0.000} C_DIS
LIN {X 104.225,Y -33.314,Z -37.053,A -90.000,B 90.000,C 0.000} C_DIS
LIN {X 104.510,Y -33.312,Z -36.928,A -90.000,B 90.000,C 0.000} C_DIS
LIN {X 105.397,Y -33.310,Z -36.555,A -90.000,B 90.000,C 0.000} C_DIS
LIN {X 106.867,Y -33.309,Z -35.970,A -90.000,B 90.000,C 0.000} C_DIS
LIN {X 107.404,Y -33.308,Z -35.767,A -90.000,B 90.000,C 0.000} C_DIS
LIN {X 107.871,Y -33.308,Z -35.598,A -90.000,B 90.000,C 0.000} C_DIS
LIN {X 108.337,Y -33.308,Z -35.443,A -90.000,B 90.000,C 0.000} C_DIS
LIN {X 108.726,Y -33.308,Z -35.338,A -90.000,B 90.000,C 0.000} C_DIS
LIN {X 108.769,Y -33.308,Z -35.328,A -90.000,B 90.000,C 0.000} C_DIS
LIN {X 109.221,Y -33.308,Z -35.225,A -90.000,B 90.000,C 0.000} C_DIS
LIN {X 109.497,Y -33.308,Z -35.161,A -90.000,B 90.000,C 0.000} C_DIS
LIN {X 109.849,Y -33.308,Z -35.071,A -90.000,B 90.000,C 0.000} C_DIS
LIN {X 110.046,Y -33.308,Z -35.016,A -90.000,B 90.000,C 0.000} C_DIS
LIN {X 110.288,Y -33.308,Z -34.941,A -90.000,B 90.000,C 0.000} C_DIS
LIN {X 110.418,Y -33.308,Z -34.896,A -90.000,B 90.000,C 0.000} C_DIS
LIN {X 110.613,Y -33.308,Z -34.819,A -90.000,B 90.000,C 0.000} C_DIS
LIN {X 110.736,Y -33.308,Z -34.759,A -90.000,B 90.000,C 0.000} C_DIS
LIN {X 110.775,Y -33.308,Z -34.736,A -90.000,B 90.000,C 0.000} C_DIS
LIN {X 110.846,Y -33.308,Z -34.687,A -90.000,B 90.000,C 0.000} C_DIS
LIN {X 110.917,Y -33.308,Z -34.758,A -90.000,B 90.000,C 0.000} C_DIS
LIN {X 111.006,Y -33.308,Z -34.821,A -90.000,B 90.000,C 0.000} C_DIS
LIN {X 111.073,Y -33.308,Z -34.861,A -90.000,B 90.000,C 0.000} C_DIS
LIN {X 111.158,Y -33.308,Z -34.905,A -90.000,B 90.000,C 0.000} C_DIS
LIN {X 111.323,Y -33.308,Z -34.982,A -90.000,B 90.000,C 0.000} C_DIS
LIN {X 111.540,Y -33.308,Z -35.072,A -90.000,B 90.000,C 0.000} C_DIS
LIN {X 111.818,Y -33.308,Z -35.173,A -90.000,B 90.000,C 0.000} C_DIS
LIN {X 112.163,Y -33.308,Z -35.288,A -90.000,B 90.000,C 0.000} C_DIS
LIN {X 112.435,Y -33.308,Z -35.371,A -90.000,B 90.000,C 0.000} C_DIS
LIN {X 112.872,Y -33.308,Z -35.502,A -90.000,B 90.000,C 0.000} C_DIS
LIN {X 113.258,Y -33.308,Z -35.612,A -90.000,B 90.000,C 0.000} C_DIS
LIN {X 113.415,Y -33.308,Z -35.653,A -90.000,B 90.000,C 0.000} C_DIS
LIN {X 113.669,Y -33.308,Z -35.713,A -90.000,B 90.000,C 0.000} C_DIS
LIN {X 113.851,Y -33.308,Z -35.747,A -90.000,B 90.000,C 0.000} C_DIS
LIN {X 113.972,Y -33.308,Z -35.763,A -90.000,B 90.000,C 0.000} C_DIS
LIN {X 114.046,Y -33.308,Z -35.765,A -90.000,B 90.000,C 0.000} C_DIS
LIN {X 114.102,Y -33.308,Z -35.757,A -90.000,B 90.000,C 0.000} C_DIS
LIN {X 114.128,Y -33.308,Z -35.808,A -90.000,B 90.000,C 0.000} C_DIS
LIN {X 114.172,Y -33.308,Z -35.867,A -90.000,B 90.000,C 0.000} C_DIS
LIN {X 114.254,Y -33.308,Z -35.958,A -90.000,B 90.000,C 0.000} C_DIS
LIN {X 114.387,Y -33.308,Z -36.087,A -90.000,B 90.000,C 0.000} C_DIS
LIN {X 114.581,Y -33.308,Z -36.261,A -90.000,B 90.000,C 0.000} C_DIS
LIN {X 114.706,Y -33.308,Z -36.366,A -90.000,B 90.000,C 0.000} C_DIS
LIN {X 115.017,Y -33.308,Z -36.618,A -90.000,B 90.000,C 0.000} C_DIS
LIN {X 115.050,Y -33.308,Z -36.644,A -90.000,B 90.000,C 0.000} C_DIS
LIN {X 115.171,Y -33.306,Z -36.736,A -90.000,B 90.000,C 0.000} C_DIS
LIN {X 115.282,Y -33.308,Z -36.825,A -90.000,B 90.000,C 0.000} C_DIS
LIN {X 115.586,Y -33.308,Z -37.050,A -90.000,B 90.000,C 0.000} C_DIS
LIN {X 115.838,Y -33.308,Z -37.225,A -90.000,B 90.000,C 0.000} C_DIS
LIN {X 116.044,Y -33.308,Z -37.356,A -90.000,B 90.000,C 0.000} C_DIS
LIN {X 116.208,Y -33.308,Z -37.450,A -90.000,B 90.000,C 0.000} C_DIS
LIN {X 116.296,Y -33.308,Z -37.495,A -90.000,B 90.000,C 0.000} C_DIS
LIN {X 116.370,Y -33.308,Z -37.528,A -90.000,B 90.000,C 0.000} C_DIS
LIN {X 116.477,Y -33.308,Z -37.567,A -90.000,B 90.000,C 0.000} C_DIS
LIN {X 116.580,Y -33.308,Z -37.586,A -90.000,B 90.000,C 0.000} C_DIS
LIN {X 116.580,Y -33.308,Z -37.676,A -90.000,B 90.000,C 0.000} C_DIS
LIN {X 116.583,Y -33.308,Z -37.724,A -90.000,B 90.000,C 0.000} C_DIS
LIN {X 116.604,Y -33.308,Z -37.865,A -90.000,B 90.000,C 0.000} C_DIS
LIN {X 116.652,Y -33.308,Z -38.077,A -90.000,B 90.000,C 0.000} C_DIS
LIN {X 116.691,Y -33.308,Z -38.215,A -90.000,B 90.000,C 0.000} C_DIS
LIN {X 116.769,Y -33.308,Z -38.467,A -90.000,B 90.000,C 0.000} C_DIS
LIN {X 116.838,Y -33.308,Z -38.667,A -90.000,B 90.000,C 0.000} C_DIS
LIN {X 116.969,Y -33.308,Z -39.021,A -90.000,B 90.000,C 0.000} C_DIS
LIN {X 117.077,Y -33.308,Z -39.295,A -90.000,B 90.000,C 0.000} C_DIS
LIN {X 117.089,Y -33.308,Z -39.324,A -90.000,B 90.000,C 0.000} C_DIS
LIN {X 117.312,Y -33.308,Z -39.862,A -90.000,B 90.000,C 0.000} C_DIS
LIN {X 117.407,Y -33.308,Z -40.079,A -90.000,B 90.000,C 0.000} C_DIS
LIN {X 117.567,Y -33.308,Z -40.422,A -90.000,B 90.000,C 0.000} C_DIS
LIN {X 117.633,Y -33.308,Z -40.553,A -90.000,B 90.000,C 0.000} C_DIS
LIN {X 117.740,Y -33.308,Z -40.746,A -90.000,B 90.000,C 0.000} C_DIS
LIN {X 117.814,Y -33.308,Z -40.864,A -90.000,B 90.000,C 0.000} C_DIS
LIN {X 117.890,Y -33.308,Z -40.959,A -90.000,B 90.000,C 0.000} C_DIS
LIN {X 117.867,Y -33.308,Z -40.987,A -90.000,B 90.000,C 0.000} C_DIS
LIN {X 117.838,Y -33.308,Z -41.040,A -90.000,B 90.000,C 0.000} C_DIS
LIN {X 117.803,Y -33.308,Z -41.145,A -90.000,B 90.000,C 0.000} C_DIS
LIN {X 117.784,Y -33.308,Z -41.224,A -90.000,B 90.000,C 0.000} C_DIS
LIN {X 117.765,Y -33.308,Z -41.322,A -90.000,B 90.000,C 0.000} C_DIS
LIN {X 117.737,Y -33.308,Z -41.514,A -90.000,B 90.000,C 0.000} C_DIS
LIN {X 117.711,Y -33.308,Z -41.765,A -90.000,B 90.000,C 0.000} C_DIS
LIN {X 117.690,Y -33.308,Z -42.083,A -90.000,B 90.000,C 0.000} C_DIS
LIN {X 117.673,Y -33.308,Z -42.478,A -90.000,B 90.000,C 0.000} C_DIS
LIN {X 117.666,Y -33.308,Z -42.788,A -90.000,B 90.000,C 0.000} C_DIS
LIN {X 117.665,Y -33.308,Z -42.838,A -90.000,B 90.000,C 0.000} C_DIS
LIN {X 117.661,Y -33.308,Z -43.386,A -90.000,B 90.000,C 0.000} C_DIS
LIN {X 117.663,Y -33.307,Z -43.608,A -90.000,B 90.000,C 0.000} C_DIS
LIN {X 117.672,Y -33.304,Z -43.961,A -90.000,B 90.000,C 0.000} C_DIS
LIN {X 117.686,Y -33.301,Z -44.209,A -90.000,B 90.000,C 0.000} C_DIS
LIN {X 117.703,Y -33.297,Z -44.370,A -90.000,B 90.000,C 0.000} C_DIS
LIN {X 117.720,Y -33.293,Z -44.464,A -90.000,B 90.000,C 0.000} C_DIS
LIN {X 117.727,Y -33.291,Z -44.491,A -90.000,B 90.000,C 0.000} C_DIS
LIN {X 117.741,Y -33.284,Z -44.525,A -90.000,B 90.000,C 0.000} C_DIS
LIN {X 117.725,Y -33.281,Z -44.538,A -90.000,B 90.000,C 0.000} C_DIS
LIN {X 117.697,Y -33.280,Z -44.576,A -90.000,B 90.000,C 0.000} C_DIS
LIN {X 117.651,Y -33.280,Z -44.660,A -90.000,B 90.000,C 0.000} C_DIS
LIN {X 117.585,Y -33.283,Z -44.808,A -90.000,B 90.000,C 0.000} C_DIS
LIN {X 117.495,Y -33.287,Z -45.040,A -90.000,B 90.000,C 0.000} C_DIS
LIN {X 117.379,Y -33.294,Z -45.374,A -90.000,B 90.000,C 0.000} C_DIS
LIN {X 117.311,Y -33.298,Z -45.585,A -90.000,B 90.000,C 0.000} C_DIS
LIN {X 117.150,Y -33.308,Z -46.109,A -90.000,B 90.000,C 0.000} C_DIS
LIN {X 117.129,Y -33.310,Z -46.181,A -90.000,B 90.000,C 0.000} C_DIS
LIN {X 117.121,Y -33.308,Z -46.207,A -90.000,B 90.000,C 0.000} C_DIS
LIN {X 116.962,Y -33.278,Z -46.755,A -90.000,B 90.000,C 0.000} C_DIS
LIN {X 116.805,Y -33.244,Z -47.332,A -90.000,B 90.000,C 0.000} C_DIS
LIN {X 116.744,Y -33.229,Z -47.580,A -90.000,B 90.000,C 0.000} C_DIS
LIN {X 116.709,Y -33.219,Z -47.742,A -90.000,B 90.000,C 0.000} C_DIS
LIN {X 116.691,Y -33.213,Z -47.863,A -90.000,B 90.000,C 0.000} C_DIS
LIN {X 116.691,Y -33.219,Z -47.895,A -90.000,B 90.000,C 0.000} C_DIS
LIN {X 116.685,Y -33.226,Z -47.898,A -90.000,B 90.000,C 0.000} C_DIS
LIN {X 116.665,Y -33.235,Z -47.917,A -90.000,B 90.000,C 0.000} C_DIS
LIN {X 116.623,Y -33.247,Z -47.971,A -90.000,B 90.000,C 0.000} C_DIS
LIN {X 116.553,Y -33.259,Z -48.078,A -90.000,B 90.000,C 0.000} C_DIS
LIN {X 116.447,Y -33.272,Z -48.258,A -90.000,B 90.000,C 0.000} C_DIS
LIN {X 116.297,Y -33.285,Z -48.529,A -90.000,B 90.000,C 0.000} C_DIS
LIN {X 116.204,Y -33.291,Z -48.705,A -90.000,B 90.000,C 0.000} C_DIS
LIN {X 115.975,Y -33.303,Z -49.148,A -90.000,B 90.000,C 0.000} C_DIS
LIN {X 115.838,Y -33.308,Z -49.420,A -90.000,B 90.000,C 0.000} C_DIS
LIN {X 115.400,Y -33.324,Z -50.296,A -90.000,B 90.000,C 0.000} C_DIS
LIN {X 115.290,Y -33.311,Z -50.516,A -90.000,B 90.000,C 0.000} C_DIS
LIN {X 115.280,Y -33.308,Z -50.537,A -90.000,B 90.000,C 0.000} C_DIS
LIN {X 115.064,Y -33.261,Z -50.969,A -90.000,B 90.000,C 0.000} C_DIS
LIN {X 115.036,Y -33.291,Z -51.025,A -90.000,B 90.000,C 0.000} C_DIS
LIN {X 114.841,Y -33.308,Z -51.405,A -90.000,B 90.000,C 0.000} C_DIS
LIN {X 114.622,Y -33.308,Z -51.838,A -90.000,B 90.000,C 0.000} C_DIS
LIN {X 114.622,Y -60.000,Z -51.838,A -90.000,B 90.000,C 0.000} C_DIS
LIN {X 94.508,Y -60.000,Z -45.193,A -90.000,B 90.000,C 0.000} C_DIS
LIN {X 94.508,Y -33.308,Z -45.193,A -90.000,B 90.000,C 0.000} C_DIS
LIN {X 94.749,Y -33.371,Z -44.883,A -90.000,B 90.000,C 0.000} C_DIS
LIN {X 94.758,Y -33.342,Z -44.770,A -90.000,B 90.000,C 0.000} C_DIS
LIN {X 94.770,Y -33.308,Z -44.652,A -90.000,B 90.000,C 0.000} C_DIS
LIN {X 94.770,Y -60.000,Z -44.652,A -90.000,B 90.000,C 0.000} C_DIS
LIN {X -21.229,Y -60.000,Z -65.803,A -90.000,B 90.000,C 0.000} C_DIS
LIN {X -21.229,Y -33.308,Z -65.803,A -90.000,B 90.000,C 0.000} C_DIS
LIN {X -20.715,Y -33.498,Z -65.504,A -90.000,B 90.000,C 0.000} C_DIS
LIN {X -20.420,Y -33.608,Z -65.342,A -90.000,B 90.000,C 0.000} C_DIS
LIN {X -20.312,Y -33.649,Z -65.286,A -90.000,B 90.000,C 0.000} C_DIS
LIN {X -20.168,Y -33.706,Z -65.215,A -90.000,B 90.000,C 0.000} C_DIS
LIN {X -20.014,Y -33.770,Z -65.147,A -90.000,B 90.000,C 0.000} C_DIS
LIN {X -19.943,Y -33.799,Z -65.117,A -90.000,B 90.000,C 0.000} C_DIS
LIN {X -19.510,Y -33.945,Z -64.949,A -90.000,B 90.000,C 0.000} C_DIS
LIN {X -19.416,Y -33.970,Z -64.914,A -90.000,B 90.000,C 0.000} C_DIS
LIN {X -18.886,Y -34.095,Z -64.728,A -90.000,B 90.000,C 0.000} C_DIS
LIN {X -18.422,Y -34.202,Z -64.544,A -90.000,B 90.000,C 0.000} C_DIS
LIN {X -18.297,Y -34.229,Z -64.500,A -90.000,B 90.000,C 0.000} C_DIS
LIN {X -18.190,Y -34.252,Z -64.466,A -90.000,B 90.000,C 0.000} C_DIS
LIN {X -17.830,Y -34.331,Z -64.362,A -90.000,B 90.000,C 0.000} C_DIS
LIN {X -17.693,Y -34.358,Z -64.325,A -90.000,B 90.000,C 0.000} C_DIS
LIN {X -17.546,Y -34.387,Z -64.291,A -90.000,B 90.000,C 0.000} C_DIS
LIN {X -17.130,Y -34.476,Z -64.216,A -90.000,B 90.000,C 0.000} C_DIS
LIN {X -16.759,Y -34.534,Z -64.156,A -90.000,B 90.000,C 0.000} C_DIS
LIN {X -16.589,Y -34.557,Z -64.130,A -90.000,B 90.000,C 0.000} C_DIS
LIN {X -16.204,Y -34.584,Z -64.075,A -90.000,B 90.000,C 0.000} C_DIS
LIN {X -15.613,Y -34.630,Z -64.008,A -90.000,B 90.000,C 0.000} C_DIS
LIN {X -15.163,Y -34.650,Z -63.890,A -90.000,B 90.000,C 0.000} C_DIS
LIN {X -15.048,Y -34.652,Z -63.865,A -90.000,B 90.000,C 0.000} C_DIS
LIN {X -14.911,Y -34.657,Z -63.840,A -90.000,B 90.000,C 0.000} C_DIS
LIN {X -14.679,Y -34.606,Z -63.598,A -90.000,B 90.000,C 0.000} C_DIS
LIN {X -14.592,Y -34.587,Z -63.506,A -90.000,B 90.000,C 0.000} C_DIS
LIN {X -14.515,Y -34.562,Z -63.428,A -90.000,B 90.000,C 0.000} C_DIS
LIN {X -14.349,Y -34.513,Z -63.270,A -90.000,B 90.000,C 0.000} C_DIS
LIN {X -14.171,Y -34.464,Z -63.110,A -90.000,B 90.000,C 0.000} C_DIS
LIN {X -13.945,Y -34.413,Z -62.931,A -90.000,B 90.000,C 0.000} C_DIS
LIN {X -13.858,Y -34.393,Z -62.870,A -90.000,B 90.000,C 0.000} C_DIS
LIN {X -13.745,Y -34.369,Z -62.795,A -90.000,B 90.000,C 0.000} C_DIS
LIN {X -13.632,Y -34.347,Z -62.725,A -90.000,B 90.000,C 0.000} C_DIS
LIN {X -13.426,Y -34.311,Z -62.609,A -90.000,B 90.000,C 0.000} C_DIS
LIN {X -13.389,Y -34.305,Z -62.589,A -90.000,B 90.000,C 0.000} C_DIS
LIN {X -13.262,Y -34.277,Z -62.525,A -90.000,B 90.000,C 0.000} C_DIS
LIN {X -13.143,Y -34.252,Z -62.470,A -90.000,B 90.000,C 0.000} C_DIS
LIN {X -12.992,Y -34.221,Z -62.404,A -90.000,B 90.000,C 0.000} C_DIS
LIN {X -12.883,Y -34.201,Z -62.360,A -90.000,B 90.000,C 0.000} C_DIS
LIN {X -12.674,Y -34.169,Z -62.290,A -90.000,B 90.000,C 0.000} C_DIS
LIN {X -12.503,Y -34.139,Z -62.240,A -90.000,B 90.000,C 0.000} C_DIS
LIN {X -12.321,Y -34.113,Z -62.196,A -90.000,B 90.000,C 0.000} C_DIS
LIN {X -11.822,Y -34.042,Z -62.080,A -90.000,B 90.000,C 0.000} C_DIS
LIN {X -11.426,Y -33.980,Z -61.993,A -90.000,B 90.000,C 0.000} C_DIS
LIN {X -11.280,Y -33.960,Z -61.964,A -90.000,B 90.000,C 0.000} C_DIS
LIN {X -10.784,Y -33.895,Z -61.878,A -90.000,B 90.000,C 0.000} C_DIS
LIN {X -10.635,Y -33.876,Z -61.857,A -90.000,B 90.000,C 0.000} C_DIS
LIN {X -9.029,Y -33.678,Z -61.681,A -90.000,B 90.000,C 0.000} C_DIS
LIN {X -8.919,Y -33.666,Z -61.671,A -90.000,B 90.000,C 0.000} C_DIS
LIN {X -8.803,Y -33.655,Z -61.664,A -90.000,B 90.000,C 0.000} C_DIS
LIN {X -8.549,Y -33.636,Z -61.655,A -90.000,B 90.000,C 0.000} C_DIS
LIN {X -8.308,Y -33.623,Z -61.655,A -90.000,B 90.000,C 0.000} C_DIS
LIN {X -7.723,Y -33.580,Z -61.659,A -90.000,B 90.000,C 0.000} C_DIS
LIN {X -6.664,Y -33.496,Z -61.672,A -90.000,B 90.000,C 0.000} C_DIS
LIN {X -6.525,Y -33.487,Z -61.677,A -90.000,B 90.000,C 0.000} C_DIS
LIN {X -5.881,Y -33.453,Z -61.711,A -90.000,B 90.000,C 0.000} C_DIS
LIN {X -5.758,Y -33.445,Z -61.715,A -90.000,B 90.000,C 0.000} C_DIS
LIN {X -5.108,Y -33.394,Z -61.743,A -90.000,B 90.000,C 0.000} C_DIS
LIN {X -4.604,Y -33.350,Z -61.769,A -90.000,B 90.000,C 0.000} C_DIS
LIN {X -3.958,Y -33.308,Z -61.795,A -90.000,B 90.000,C 0.000} C_DIS
LIN {X -3.958,Y -60.000,Z -61.795,A -90.000,B 90.000,C 0.000} C_DIS
LIN {X -20.086,Y -60.000,Z -63.141,A -90.000,B 90.000,C 0.000} C_DIS
LIN {X -20.086,Y -33.308,Z -63.141,A -90.000,B 90.000,C 0.000} C_DIS
LIN {X -19.847,Y -33.396,Z -63.046,A -90.000,B 90.000,C 0.000} C_DIS
LIN {X -19.704,Y -33.445,Z -62.991,A -90.000,B 90.000,C 0.000} C_DIS
LIN {X -19.563,Y -33.489,Z -62.938,A -90.000,B 90.000,C 0.000} C_DIS
LIN {X -19.404,Y -33.532,Z -62.879,A -90.000,B 90.000,C 0.000} C_DIS
LIN {X -19.287,Y -33.560,Z -62.832,A -90.000,B 90.000,C 0.000} C_DIS
LIN {X -19.005,Y -33.603,Z -62.727,A -90.000,B 90.000,C 0.000} C_DIS
LIN {X -18.817,Y -33.627,Z -62.665,A -90.000,B 90.000,C 0.000} C_DIS
LIN {X -18.599,Y -33.653,Z -62.602,A -90.000,B 90.000,C 0.000} C_DIS
LIN {X -18.332,Y -33.687,Z -62.533,A -90.000,B 90.000,C 0.000} C_DIS
LIN {X -18.068,Y -33.718,Z -62.467,A -90.000,B 90.000,C 0.000} C_DIS
LIN {X -17.842,Y -33.748,Z -62.420,A -90.000,B 90.000,C 0.000} C_DIS
LIN {X -17.753,Y -33.760,Z -62.403,A -90.000,B 90.000,C 0.000} C_DIS
LIN {X -16.790,Y -33.904,Z -62.250,A -90.000,B 90.000,C 0.000} C_DIS
LIN {X -16.614,Y -33.929,Z -62.221,A -90.000,B 90.000,C 0.000} C_DIS
LIN {X -16.336,Y -33.957,Z -62.180,A -90.000,B 90.000,C 0.000} C_DIS
LIN {X -16.259,Y -33.963,Z -62.171,A -90.000,B 90.000,C 0.000} C_DIS
LIN {X -16.011,Y -33.976,Z -62.145,A -90.000,B 90.000,C 0.000} C_DIS
LIN {X -15.926,Y -33.977,Z -62.137,A -90.000,B 90.000,C 0.000} C_DIS
LIN {X -15.836,Y -33.948,Z -62.053,A -90.000,B 90.000,C 0.000} C_DIS
LIN {X -15.673,Y -33.882,Z -61.909,A -90.000,B 90.000,C 0.000} C_DIS
LIN {X -15.466,Y -33.802,Z -61.737,A -90.000,B 90.000,C 0.000} C_DIS
LIN {X -15.155,Y -33.697,Z -61.508,A -90.000,B 90.000,C 0.000} C_DIS
LIN {X -14.948,Y -33.635,Z -61.373,A -90.000,B 90.000,C 0.000} C_DIS
LIN {X -14.881,Y -33.614,Z -61.332,A -90.000,B 90.000,C 0.000} C_DIS
LIN {X -14.707,Y -33.564,Z -61.231,A -90.000,B 90.000,C 0.000} C_DIS
LIN {X -14.460,Y -33.499,Z -61.101,A -90.000,B 90.000,C 0.000} C_DIS
LIN {X -14.369,Y -33.474,Z -61.056,A -90.000,B 90.000,C 0.000} C_DIS
LIN {X -14.157,Y -33.415,Z -60.958,A -90.000,B 90.000,C 0.000} C_DIS
LIN {X -13.893,Y -33.347,Z -60.847,A -90.000,B 90.000,C 0.000} C_DIS
LIN {X -13.815,Y -33.328,Z -60.816,A -90.000,B 90.000,C 0.000} C_DIS
LIN {X -13.725,Y -33.308,Z -60.781,A -90.000,B 90.000,C 0.000} C_DIS
LIN {X -13.725,Y -60.000,Z -60.781,A -90.000,B 90.000,C 0.000} C_DIS
LIN {X -41.557,Y -60.000,Z -103.914,A -90.000,B 90.000,C 0.000} C_DIS
LIN {X -41.557,Y -33.308,Z -103.914,A -90.000,B 90.000,C 0.000} C_DIS
LIN {X -41.567,Y -33.379,Z -103.701,A -90.000,B 90.000,C 0.000} C_DIS
LIN {X -41.587,Y -33.528,Z -103.292,A -90.000,B 90.000,C 0.000} C_DIS
LIN {X -41.594,Y -33.622,Z -103.041,A -90.000,B 90.000,C 0.000} C_DIS
LIN {X -41.710,Y -33.622,Z -102.889,A -90.000,B 90.000,C 0.000} C_DIS
LIN {X -42.388,Y -33.626,Z -101.973,A -90.000,B 90.000,C 0.000} C_DIS
LIN {X -42.786,Y -33.631,Z -101.411,A -90.000,B 90.000,C 0.000} C_DIS
LIN {X -43.482,Y -33.633,Z -100.414,A -90.000,B 90.000,C 0.000} C_DIS
LIN {X -43.739,Y -33.638,Z -100.035,A -90.000,B 90.000,C 0.000} C_DIS
LIN {X -44.021,Y -33.654,Z -99.590,A -90.000,B 90.000,C 0.000} C_DIS
LIN {X -44.755,Y -33.678,Z -98.417,A -90.000,B 90.000,C 0.000} C_DIS
LIN {X -45.351,Y -33.704,Z -97.445,A -90.000,B 90.000,C 0.000} C_DIS
LIN {X -45.763,Y -33.734,Z -96.730,A -90.000,B 90.000,C 0.000} C_DIS
LIN {X -45.981,Y -33.741,Z -96.329,A -90.000,B 90.000,C 0.000} C_DIS
LIN {X -46.658,Y -33.741,Z -95.073,A -90.000,B 90.000,C 0.000} C_DIS
LIN {X -46.920,Y -33.745,Z -94.567,A -90.000,B 90.000,C 0.000} C_DIS
LIN {X -47.299,Y -33.744,Z -93.828,A -90.000,B 90.000,C 0.000} C_DIS
LIN {X -47.604,Y -33.754,Z -93.182,A -90.000,B 90.000,C 0.000} C_DIS
LIN {X -47.655,Y -33.756,Z -93.067,A -90.000,B 90.000,C 0.000} C_DIS
LIN {X -47.868,Y -33.761,Z -92.566,A -90.000,B 90.000,C 0.000} C_DIS
LIN {X -48.294,Y -33.751,Z -91.547,A -90.000,B 90.000,C 0.000} C_DIS
LIN {X -48.500,Y -33.744,Z -91.037,A -90.000,B 90.000,C 0.000} C_DIS
LIN {X -48.514,Y -33.744,Z -91.002,A -90.000,B 90.000,C 0.000} C_DIS
LIN {X -48.819,Y -33.740,Z -90.202,A -90.000,B 90.000,C 0.000} C_DIS
LIN {X -49.033,Y -33.739,Z -89.626,A -90.000,B 90.000,C 0.000} C_DIS
LIN {X -49.065,Y -33.740,Z -89.532,A -90.000,B 90.000,C 0.000} C_DIS
LIN {X -49.256,Y -33.743,Z -88.932,A -90.000,B 90.000,C 0.000} C_DIS
LIN {X -49.474,Y -33.751,Z -88.160,A -90.000,B 90.000,C 0.000} C_DIS
LIN {X -49.504,Y -33.752,Z -88.047,A -90.000,B 90.000,C 0.000} C_DIS
LIN {X -49.913,Y -33.794,Z -86.382,A -90.000,B 90.000,C 0.000} C_DIS
LIN {X -50.040,Y -33.801,Z -85.852,A -90.000,B 90.000,C 0.000} C_DIS
LIN {X -50.117,Y -33.803,Z -85.541,A -90.000,B 90.000,C 0.000} C_DIS
LIN {X -50.136,Y -33.804,Z -85.457,A -90.000,B 90.000,C 0.000} C_DIS
LIN {X -50.176,Y -33.808,Z -85.254,A -90.000,B 90.000,C 0.000} C_DIS
LIN {X -50.213,Y -33.816,Z -85.026,A -90.000,B 90.000,C 0.000} C_DIS
LIN {X -50.258,Y -33.829,Z -84.714,A -90.000,B 90.000,C 0.000} C_DIS
LIN {X -50.297,Y -33.841,Z -84.427,A -90.000,B 90.000,C 0.000} C_DIS
LIN {X -50.402,Y -33.885,Z -83.515,A -90.000,B 90.000,C 0.000} C_DIS
LIN {X -50.480,Y -33.899,Z -82.769,A -90.000,B 90.000,C 0.000} C_DIS
LIN {X -50.510,Y -33.908,Z -82.476,A -90.000,B 90.000,C 0.000} C_DIS
LIN {X -50.520,Y -33.922,Z -82.224,A -90.000,B 90.000,C 0.000} C_DIS
LIN {X -50.522,Y -33.930,Z -82.086,A -90.000,B 90.000,C 0.000} C_DIS
LIN {X -50.513,Y -33.965,Z -81.623,A -90.000,B 90.000,C 0.000} C_DIS
LIN {X -50.507,Y -33.980,Z -81.377,A -90.000,B 90.000,C 0.000} C_DIS
LIN {X -50.497,Y -33.993,Z -81.036,A -90.000,B 90.000,C 0.000} C_DIS
LIN {X -50.446,Y -34.045,Z -79.850,A -90.000,B 90.000,C 0.000} C_DIS
LIN {X -50.439,Y -34.051,Z -79.741,A -90.000,B 90.000,C 0.000} C_DIS
LIN {X -50.431,Y -34.057,Z -79.649,A -90.000,B 90.000,C 0.000} C_DIS
LIN {X -50.416,Y -34.061,Z -79.508,A -90.000,B 90.000,C 0.000} C_DIS
LIN {X -50.268,Y -34.103,Z -78.513,A -90.000,B 90.000,C 0.000} C_DIS
LIN {X -50.230,Y -34.114,Z -78.280,A -90.000,B 90.000,C 0.000} C_DIS
LIN {X -50.127,Y -34.139,Z -77.722,A -90.000,B 90.000,C 0.000} C_DIS
LIN {X -50.034,Y -34.152,Z -77.241,A -90.000,B 90.000,C 0.000} C_DIS
LIN {X -49.995,Y -34.158,Z -77.066,A -90.000,B 90.000,C 0.000} C_DIS
LIN {X -49.799,Y -34.192,Z -76.290,A -90.000,B 90.000,C 0.000} C_DIS
LIN {X -49.769,Y -34.196,Z -76.176,A -90.000,B 90.000,C 0.000} C_DIS
LIN {X -49.671,Y -34.212,Z -75.789,A -90.000,B 90.000,C 0.000} C_DIS
LIN {X -49.612,Y -34.217,Z -75.572,A -90.000,B 90.000,C 0.000} C_DIS
LIN {X -49.514,Y -34.227,Z -75.246,A -90.000,B 90.000,C 0.000} C_DIS
LIN {X -49.381,Y -34.242,Z -74.838,A -90.000,B 90.000,C 0.000} C_DIS
LIN {X -49.213,Y -34.263,Z -74.348,A -90.000,B 90.000,C 0.000} C_DIS
LIN {X -48.919,Y -34.278,Z -73.518,A -90.000,B 90.000,C 0.000} C_DIS
LIN {X -48.845,Y -34.283,Z -73.330,A -90.000,B 90.000,C 0.000} C_DIS
LIN {X -48.585,Y -34.303,Z -72.717,A -90.000,B 90.000,C 0.000} C_DIS
LIN {X -48.197,Y -34.317,Z -71.805,A -90.000,B 90.000,C 0.000} C_DIS
LIN {X -48.050,Y -34.326,Z -71.494,A -90.000,B 90.000,C 0.000} C_DIS
LIN {X -47.948,Y -34.330,Z -71.284,A -90.000,B 90.000,C 0.000} C_DIS
LIN {X -47.842,Y -34.328,Z -71.073,A -90.000,B 90.000,C 0.000} C_DIS
LIN {X -47.652,Y -34.328,Z -70.729,A -90.000,B 90.000,C 0.000} C_DIS
LIN {X -47.232,Y -34.336,Z -70.024,A -90.000,B 90.000,C 0.000} C_DIS
LIN {X -47.069,Y -34.336,Z -69.756,A -90.000,B 90.000,C 0.000} C_DIS
LIN {X -47.009,Y -34.334,Z -69.665,A -90.000,B 90.000,C 0.000} C_DIS
LIN {X -46.530,Y -34.306,Z -68.954,A -90.000,B 90.000,C 0.000} C_DIS
LIN {X -46.472,Y -34.304,Z -68.872,A -90.000,B 90.000,C 0.000} C_DIS
LIN {X -46.400,Y -34.302,Z -68.777,A -90.000,B 90.000,C 0.000} C_DIS
LIN {X -46.254,Y -34.299,Z -68.600,A -90.000,B 90.000,C 0.000} C_DIS
LIN {X -46.007,Y -34.295,Z -68.322,A -90.000,B 90.000,C 0.000} C_DIS
LIN {X -45.905,Y -34.294,Z -68.213,A -90.000,B 90.000,C 0.000} C_DIS
LIN {X -45.756,Y -34.284,Z -68.058,A -90.000,B 90.000,C 0.000} C_DIS
LIN {X -45.451,Y -34.259,Z -67.745,A -90.000,B 90.000,C 0.000} C_DIS
LIN {X -45.180,Y -34.240,Z -67.483,A -90.000,B 90.000,C 0.000} C_DIS
LIN {X -44.483,Y -34.181,Z -66.814,A -90.000,B 90.000,C 0.000} C_DIS
LIN {X -44.202,Y -34.164,Z -66.576,A -90.000,B 90.000,C 0.000} C_DIS
LIN {X -44.115,Y -34.158,Z -66.509,A -90.000,B 90.000,C 0.000} C_DIS
LIN {X -44.010,Y -34.151,Z -66.433,A -90.000,B 90.000,C 0.000} C_DIS
LIN {X -43.815,Y -34.128,Z -66.299,A -90.000,B 90.000,C 0.000} C_DIS
LIN {X -43.457,Y -34.092,Z -66.073,A -90.000,B 90.000,C 0.000} C_DIS
LIN {X -43.254,Y -34.074,Z -65.957,A -90.000,B 90.000,C 0.000} C_DIS
LIN {X -42.101,Y -33.991,Z -65.344,A -90.000,B 90.000,C 0.000} C_DIS
LIN {X -41.906,Y -33.975,Z -65.242,A -90.000,B 90.000,C 0.000} C_DIS
LIN {X -41.484,Y -33.939,Z -65.041,A -90.000,B 90.000,C 0.000} C_DIS
LIN {X -41.274,Y -33.918,Z -64.943,A -90.000,B 90.000,C 0.000} C_DIS
LIN {X -40.509,Y -33.826,Z -64.594,A -90.000,B 90.000,C 0.000} C_DIS
LIN {X -40.428,Y -33.817,Z -64.560,A -90.000,B 90.000,C 0.000} C_DIS
LIN {X -40.344,Y -33.810,Z -64.528,A -90.000,B 90.000,C 0.000} C_DIS
LIN {X -40.070,Y -33.790,Z -64.432,A -90.000,B 90.000,C 0.000} C_DIS
LIN {X -40.022,Y -33.785,Z -64.416,A -90.000,B 90.000,C 0.000} C_DIS
LIN {X -39.924,Y -33.777,Z -64.388,A -90.000,B 90.000,C 0.000} C_DIS
LIN {X -39.516,Y -33.750,Z -64.281,A -90.000,B 90.000,C 0.000} C_DIS
LIN {X -38.555,Y -33.700,Z -64.059,A -90.000,B 90.000,C 0.000} C_DIS
LIN {X -38.398,Y -33.689,Z -64.027,A -90.000,B 90.000,C 0.000} C_DIS
LIN {X -38.327,Y -33.685,Z -64.014,A -90.000,B 90.000,C 0.000} C_DIS
LIN {X -38.031,Y -33.670,Z -63.968,A -90.000,B 90.000,C 0.000} C_DIS
LIN {X -37.048,Y -33.621,Z -63.822,A -90.000,B 90.000,C 0.000} C_DIS
LIN {X -36.807,Y -33.612,Z -63.793,A -90.000,B 90.000,C 0.000} C_DIS
LIN {X -36.666,Y -33.605,Z -63.779,A -90.000,B 90.000,C 0.000} C_DIS
LIN {X -35.268,Y -33.514,Z -63.650,A -90.000,B 90.000,C 0.000} C_DIS
LIN {X -34.830,Y -33.474,Z -63.619,A -90.000,B 90.000,C 0.000} C_DIS
LIN {X -34.642,Y -33.459,Z -63.610,A -90.000,B 90.000,C 0.000} C_DIS
LIN {X -34.439,Y -33.447,Z -63.608,A -90.000,B 90.000,C 0.000} C_DIS
LIN {X -33.496,Y -33.402,Z -63.616,A -90.000,B 90.000,C 0.000} C_DIS
LIN {X -33.098,Y -33.380,Z -63.622,A -90.000,B 90.000,C 0.000} C_DIS
LIN {X -32.614,Y -33.340,Z -63.636,A -90.000,B 90.000,C 0.000} C_DIS
LIN {X -32.515,Y -33.333,Z -63.641,A -90.000,B 90.000,C 0.000} C_DIS
LIN {X -32.085,Y -33.308,Z -63.673,A -90.000,B 90.000,C 0.000} C_DIS
LIN {X -32.085,Y -60.000,Z -63.673,A -90.000,B 90.000,C 0.000} C_DIS
LIN {X -52.384,Y -60.000,Z -81.172,A -90.000,B 90.000,C 0.000} C_DIS
LIN {X -52.384,Y -33.308,Z -81.172,A -90.000,B 90.000,C 0.000} C_DIS
LIN {X -52.376,Y -33.333,Z -80.830,A -90.000,B 90.000,C 0.000} C_DIS
LIN {X -52.358,Y -33.375,Z -80.279,A -90.000,B 90.000,C 0.000} C_DIS
LIN {X -52.347,Y -33.391,Z -79.991,A -90.000,B 90.000,C 0.000} C_DIS
LIN {X -52.329,Y -33.408,Z -79.628,A -90.000,B 90.000,C 0.000} C_DIS
LIN {X -52.316,Y -33.418,Z -79.457,A -90.000,B 90.000,C 0.000} C_DIS
LIN {X -52.301,Y -33.428,Z -79.295,A -90.000,B 90.000,C 0.000} C_DIS
LIN {X -52.291,Y -33.435,Z -79.203,A -90.000,B 90.000,C 0.000} C_DIS
LIN {X -52.192,Y -33.494,Z -78.474,A -90.000,B 90.000,C 0.000} C_DIS
LIN {X -52.148,Y -33.510,Z -78.177,A -90.000,B 90.000,C 0.000} C_DIS
LIN {X -52.101,Y -33.527,Z -77.886,A -90.000,B 90.000,C 0.000} C_DIS
LIN {X -51.931,Y -33.582,Z -76.950,A -90.000,B 90.000,C 0.000} C_DIS
LIN {X -51.904,Y -33.589,Z -76.810,A -90.000,B 90.000,C 0.000} C_DIS
LIN {X -51.852,Y -33.602,Z -76.572,A -90.000,B 90.000,C 0.000} C_DIS
LIN {X -51.604,Y -33.664,Z -75.573,A -90.000,B 90.000,C 0.000} C_DIS
LIN {X -51.477,Y -33.687,Z -75.082,A -90.000,B 90.000,C 0.000} C_DIS
LIN {X -51.367,Y -33.708,Z -74.700,A -90.000,B 90.000,C 0.000} C_DIS
LIN {X -51.204,Y -33.738,Z -74.188,A -90.000,B 90.000,C 0.000} C_DIS
LIN {X -51.143,Y -33.750,Z -74.006,A -90.000,B 90.000,C 0.000} C_DIS
LIN {X -50.744,Y -33.799,Z -72.853,A -90.000,B 90.000,C 0.000} C_DIS
LIN {X -50.653,Y -33.811,Z -72.619,A -90.000,B 90.000,C 0.000} C_DIS
LIN {X -50.043,Y -33.858,Z -71.170,A -90.000,B 90.000,C 0.000} C_DIS
LIN {X -49.952,Y -33.861,Z -70.961,A -90.000,B 90.000,C 0.000} C_DIS
LIN {X -49.760,Y -33.870,Z -70.558,A -90.000,B 90.000,C 0.000} C_DIS
LIN {X -49.582,Y -33.872,Z -70.200,A -90.000,B 90.000,C 0.000} C_DIS
LIN {X -49.450,Y -33.875,Z -69.956,A -90.000,B 90.000,C 0.000} C_DIS
LIN {X -49.323,Y -33.875,Z -69.728,A -90.000,B 90.000,C 0.000} C_DIS
LIN {X -48.911,Y -33.877,Z -69.039,A -90.000,B 90.000,C 0.000} C_DIS
LIN {X -48.700,Y -33.864,Z -68.699,A -90.000,B 90.000,C 0.000} C_DIS
LIN {X -48.517,Y -33.854,Z -68.425,A -90.000,B 90.000,C 0.000} C_DIS
LIN {X -48.101,Y -33.825,Z -67.813,A -90.000,B 90.000,C 0.000} C_DIS
LIN {X -47.985,Y -33.819,Z -67.657,A -90.000,B 90.000,C 0.000} C_DIS
LIN {X -47.932,Y -33.817,Z -67.587,A -90.000,B 90.000,C 0.000} C_DIS
LIN {X -47.781,Y -33.802,Z -67.408,A -90.000,B 90.000,C 0.000} C_DIS
LIN {X -47.683,Y -33.792,Z -67.296,A -90.000,B 90.000,C 0.000} C_DIS
LIN {X -47.487,Y -33.772,Z -67.082,A -90.000,B 90.000,C 0.000} C_DIS
LIN {X -47.355,Y -33.758,Z -66.943,A -90.000,B 90.000,C 0.000} C_DIS
LIN {X -46.807,Y -33.704,Z -66.383,A -90.000,B 90.000,C 0.000} C_DIS
LIN {X -46.387,Y -33.670,Z -65.980,A -90.000,B 90.000,C 0.000} C_DIS
LIN {X -46.226,Y -33.649,Z -65.828,A -90.000,B 90.000,C 0.000} C_DIS
LIN {X -45.828,Y -33.572,Z -65.465,A -90.000,B 90.000,C 0.000} C_DIS
LIN {X -45.733,Y -33.556,Z -65.383,A -90.000,B 90.000,C 0.000} C_DIS
LIN {X -45.447,Y -33.514,Z -65.152,A -90.000,B 90.000,C 0.000} C_DIS
LIN {X -45.294,Y -33.494,Z -65.036,A -90.000,B 90.000,C 0.000} C_DIS
LIN {X -45.249,Y -33.489,Z -65.004,A -90.000,B 90.000,C 0.000} C_DIS
LIN {X -44.957,Y -33.457,Z -64.801,A -90.000,B 90.000,C 0.000} C_DIS
LIN {X -44.825,Y -33.444,Z -64.713,A -90.000,B 90.000,C 0.000} C_DIS
LIN {X -44.687,Y -33.428,Z -64.627,A -90.000,B 90.000,C 0.000} C_DIS
LIN {X -44.501,Y -33.404,Z -64.512,A -90.000,B 90.000,C 0.000} C_DIS
LIN {X -44.208,Y -33.370,Z -64.346,A -90.000,B 90.000,C 0.000} C_DIS
LIN {X -43.683,Y -33.308,Z -64.077,A -90.000,B 90.000,C 0.000} C_DIS
LIN {X -43.683,Y -60.000,Z -64.077,A -90.000,B 90.000,C 0.000} C_DIS
LIN {X -52.758,Y -60.000,Z -72.729,A -90.000,B 90.000,C 0.000} C_DIS
LIN {X -52.758,Y -33.308,Z -72.729,A -90.000,B 90.000,C 0.000} C_DIS
LIN {X -52.550,Y -33.332,Z -72.134,A -90.000,B 90.000,C 0.000} C_DIS
LIN {X -52.441,Y -33.346,Z -71.851,A -90.000,B 90.000,C 0.000} C_DIS
LIN {X -52.240,Y -33.381,Z -71.363,A -90.000,B 90.000,C 0.000} C_DIS
LIN {X -51.797,Y -33.411,Z -70.317,A -90.000,B 90.000,C 0.000} C_DIS
LIN {X -51.696,Y -33.425,Z -70.084,A -90.000,B 90.000,C 0.000} C_DIS
LIN {X -51.594,Y -33.432,Z -69.868,A -90.000,B 90.000,C 0.000} C_DIS
LIN {X -51.329,Y -33.429,Z -69.332,A -90.000,B 90.000,C 0.000} C_DIS
LIN {X -51.154,Y -33.431,Z -69.007,A -90.000,B 90.000,C 0.000} C_DIS
LIN {X -50.996,Y -33.434,Z -68.725,A -90.000,B 90.000,C 0.000} C_DIS
LIN {X -50.803,Y -33.437,Z -68.401,A -90.000,B 90.000,C 0.000} C_DIS
LIN {X -50.573,Y -33.419,Z -68.025,A -90.000,B 90.000,C 0.000} C_DIS
LIN {X -50.361,Y -33.404,Z -67.685,A -90.000,B 90.000,C 0.000} C_DIS
LIN {X -50.110,Y -33.392,Z -67.307,A -90.000,B 90.000,C 0.000} C_DIS
LIN {X -49.915,Y -33.380,Z -67.018,A -90.000,B 90.000,C 0.000} C_DIS
LIN {X -49.718,Y -33.350,Z -66.737,A -90.000,B 90.000,C 0.000} C_DIS
LIN {X -49.553,Y -33.326,Z -66.517,A -90.000,B 90.000,C 0.000} C_DIS
LIN {X -49.407,Y -33.308,Z -66.335,A -90.000,B 90.000,C 0.000} C_DIS
LIN {X -49.407,Y -60.000,Z -66.335,A -90.000,B 90.000,C 0.000} C_DIS
LIN {X 9.579,Y -60.000,Z -172.040,A -90.000,B 90.000,C 0.000} C_DIS
LIN {X 9.579,Y -33.308,Z -172.040,A -90.000,B 90.000,C 0.000} C_DIS
LIN {X 9.614,Y -33.313,Z -172.000,A -90.000,B 90.000,C 0.000} C_DIS
LIN {X 10.206,Y -33.363,Z -171.200,A -90.000,B 90.000,C 0.000} C_DIS
LIN {X 10.295,Y -33.370,Z -171.084,A -90.000,B 90.000,C 0.000} C_DIS
LIN {X 10.950,Y -33.431,Z -170.264,A -90.000,B 90.000,C 0.000} C_DIS
LIN {X 11.148,Y -33.475,Z -169.995,A -90.000,B 90.000,C 0.000} C_DIS
LIN {X 12.013,Y -33.627,Z -168.515,A -90.000,B 90.000,C 0.000} C_DIS
LIN {X 12.163,Y -33.631,Z -168.089,A -90.000,B 90.000,C 0.000} C_DIS
LIN {X 12.211,Y -33.633,Z -167.960,A -90.000,B 90.000,C 0.000} C_DIS
LIN {X 12.525,Y -33.732,Z -167.001,A -90.000,B 90.000,C 0.000} C_DIS
LIN {X 12.532,Y -33.725,Z -166.813,A -90.000,B 90.000,C 0.000} C_DIS
LIN {X 12.554,Y -33.719,Z -166.211,A -90.000,B 90.000,C 0.000} C_DIS
LIN {X 12.542,Y -33.711,Z -166.125,A -90.000,B 90.000,C 0.000} C_DIS
LIN {X 12.428,Y -33.683,Z -165.419,A -90.000,B 90.000,C 0.000} C_DIS
LIN {X 12.387,Y -33.675,Z -165.109,A -90.000,B 90.000,C 0.000} C_DIS
LIN {X 12.361,Y -33.670,Z -164.900,A -90.000,B 90.000,C 0.000} C_DIS
LIN {X 12.351,Y -33.670,Z -164.822,A -90.000,B 90.000,C 0.000} C_DIS
LIN {X 12.270,Y -33.660,Z -164.449,A -90.000,B 90.000,C 0.000} C_DIS
LIN {X 12.205,Y -33.656,Z -164.154,A -90.000,B 90.000,C 0.000} C_DIS
LIN {X 12.102,Y -33.633,Z -163.870,A -90.000,B 90.000,C 0.000} C_DIS
LIN {X 12.031,Y -33.620,Z -163.649,A -90.000,B 90.000,C 0.000} C_DIS
LIN {X 11.994,Y -33.619,Z -163.535,A -90.000,B 90.000,C 0.000} C_DIS
LIN {X 11.774,Y -33.619,Z -162.769,A -90.000,B 90.000,C 0.000} C_DIS
LIN {X 11.554,Y -33.597,Z -162.170,A -90.000,B 90.000,C 0.000} C_DIS
LIN {X 11.393,Y -33.598,Z -161.744,A -90.000,B 90.000,C 0.000} C_DIS
LIN {X 11.325,Y -33.604,Z -161.570,A -90.000,B 90.000,C 0.000} C_DIS
LIN {X 11.287,Y -33.609,Z -161.472,A -90.000,B 90.000,C 0.000} C_DIS
LIN {X 10.987,Y -33.634,Z -160.748,A -90.000,B 90.000,C 0.000} C_DIS
LIN {X 10.922,Y -33.635,Z -160.621,A -90.000,B 90.000,C 0.000} C_DIS
LIN {X 10.844,Y -33.639,Z -160.457,A -90.000,B 90.000,C 0.000} C_DIS
LIN {X 10.605,Y -33.657,Z -159.924,A -90.000,B 90.000,C 0.000} C_DIS
LIN {X 10.345,Y -33.722,Z -159.394,A -90.000,B 90.000,C 0.000} C_DIS
LIN {X 10.313,Y -33.731,Z -159.325,A -90.000,B 90.000,C 0.000} C_DIS
LIN {X 10.234,Y -33.748,Z -159.155,A -90.000,B 90.000,C 0.000} C_DIS
LIN {X 10.103,Y -33.764,Z -158.921,A -90.000,B 90.000,C 0.000} C_DIS
LIN {X 9.726,Y -33.819,Z -158.205,A -90.000,B 90.000,C 0.000} C_DIS
LIN {X 9.590,Y -33.869,Z -157.970,A -90.000,B 90.000,C 0.000} C_DIS
LIN {X 9.267,Y -33.967,Z -157.368,A -90.000,B 90.000,C 0.000} C_DIS
LIN {X 9.154,Y -33.984,Z -157.207,A -90.000,B 90.000,C 0.000} C_DIS
LIN {X 8.411,Y -33.777,Z -157.222,A -90.000,B 90.000,C 0.000} C_DIS
LIN {X 8.132,Y -33.700,Z -157.224,A -90.000,B 90.000,C 0.000} C_DIS
LIN {X 7.607,Y -33.557,Z -157.224,A -90.000,B 90.000,C 0.000} C_DIS
LIN {X 7.402,Y -33.502,Z -157.217,A -90.000,B 90.000,C 0.000} C_DIS
LIN {X 7.119,Y -33.431,Z -157.197,A -90.000,B 90.000,C 0.000} C_DIS
LIN {X 6.865,Y -33.384,Z -157.185,A -90.000,B 90.000,C 0.000} C_DIS
LIN {X 6.697,Y -33.355,Z -157.173,A -90.000,B 90.000,C 0.000} C_DIS
LIN {X 6.432,Y -33.308,Z -157.147,A -90.000,B 90.000,C 0.000} C_DIS
LIN {X 6.432,Y -60.000,Z -157.147,A -90.000,B 90.000,C 0.000} C_DIS
LIN {X -96.739,Y -60.000,Z -243.561,A -90.000,B 90.000,C 0.000} C_DIS
LIN {X -96.739,Y -33.389,Z -243.561,A -90.000,B 90.000,C 0.000} C_DIS
LIN {X -96.709,Y -33.341,Z -243.480,A -90.000,B 90.000,C 0.000} C_DIS
LIN {X -96.685,Y -33.308,Z -243.424,A -90.000,B 90.000,C 0.000} C_DIS
LIN {X -96.679,Y -33.306,Z -243.408,A -90.000,B 90.000,C 0.000} C_DIS
LIN {X -96.676,Y -33.298,Z -243.395,A -90.000,B 90.000,C 0.000} C_DIS
LIN {X -96.676,Y -33.290,Z -243.386,A -90.000,B 90.000,C 0.000} C_DIS
LIN {X -96.683,Y -33.279,Z -243.376,A -90.000,B 90.000,C 0.000} C_DIS
LIN {X -96.698,Y -33.271,Z -243.378,A -90.000,B 90.000,C 0.000} C_DIS
LIN {X -96.734,Y -33.266,Z -243.397,A -90.000,B 90.000,C 0.000} C_DIS
LIN {X -96.794,Y -33.270,Z -243.443,A -90.000,B 90.000,C 0.000} C_DIS
LIN {X -96.884,Y -33.287,Z -243.527,A -90.000,B 90.000,C 0.000} C_DIS
LIN {X -96.922,Y -33.300,Z -243.570,A -90.000,B 90.000,C 0.000} C_DIS
LIN {X -96.929,Y -33.307,Z -243.583,A -90.000,B 90.000,C 0.000} C_DIS
LIN {X -96.926,Y -33.312,Z -243.587,A -90.000,B 90.000,C 0.000} C_DIS
LIN {X -96.920,Y -33.314,Z -243.585,A -90.000,B 90.000,C 0.000} C_DIS
LIN {X -96.911,Y -33.315,Z -243.580,A -90.000,B 90.000,C 0.000} C_DIS
LIN {X -96.881,Y -33.308,Z -243.561,A -90.000,B 90.000,C 0.000} C_DIS
LIN {X -91.603,Y -33.308,Z -239.868,A -90.000,B 90.000,C 0.000} C_DIS
LIN {X -90.107,Y -33.308,Z -238.815,A -90.000,B 90.000,C 0.000} C_DIS
LIN {X -89.804,Y -33.308,Z -238.608,A -90.000,B 90.000,C 0.000} C_DIS
LIN {X -89.694,Y -33.308,Z -238.535,A -90.000,B 90.000,C 0.000} C_DIS
LIN {X -85.913,Y -33.308,Z -236.074,A -90.000,B 90.000,C 0.000} C_DIS
LIN {X -81.593,Y -33.308,Z -233.237,A -90.000,B 90.000,C 0.000} C_DIS
LIN {X -79.393,Y -33.308,Z -231.906,A -90.000,B 90.000,C 0.000} C_DIS
LIN {X -73.176,Y -33.308,Z -228.125,A -90.000,B 90.000,C 0.000} C_DIS
LIN {X -72.554,Y -33.308,Z -227.778,A -90.000,B 90.000,C 0.000} C_DIS
LIN {X -66.820,Y -33.308,Z -224.614,A -90.000,B 90.000,C 0.000} C_DIS
LIN {X -64.604,Y -33.308,Z -223.422,A -90.000,B 90.000,C 0.000} C_DIS
LIN {X -64.277,Y -33.308,Z -223.254,A -90.000,B 90.000,C 0.000} C_DIS
LIN {X -63.086,Y -33.308,Z -222.648,A -90.000,B 90.000,C 0.000} C_DIS
LIN {X -55.740,Y -33.308,Z -218.925,A -90.000,B 90.000,C 0.000} C_DIS
LIN {X -50.003,Y -33.308,Z -216.079,A -90.000,B 90.000,C 0.000} C_DIS
LIN {X -47.803,Y -33.308,Z -214.995,A -90.000,B 90.000,C 0.000} C_DIS
LIN {X -44.144,Y -33.308,Z -213.164,A -90.000,B 90.000,C 0.000} C_DIS
LIN {X -41.005,Y -33.308,Z -211.615,A -90.000,B 90.000,C 0.000} C_DIS
LIN {X -36.783,Y -33.308,Z -209.417,A -90.000,B 90.000,C 0.000} C_DIS
LIN {X -35.373,Y -33.308,Z -208.666,A -90.000,B 90.000,C 0.000} C_DIS
LIN {X -33.168,Y -33.308,Z -207.432,A -90.000,B 90.000,C 0.000} C_DIS
LIN {X -30.586,Y -33.308,Z -205.959,A -90.000,B 90.000,C 0.000} C_DIS
LIN {X -29.469,Y -33.308,Z -205.282,A -90.000,B 90.000,C 0.000} C_DIS
LIN {X -26.495,Y -33.308,Z -203.450,A -90.000,B 90.000,C 0.000} C_DIS
LIN {X -26.100,Y -33.308,Z -203.190,A -90.000,B 90.000,C 0.000} C_DIS
LIN {X -23.033,Y -33.308,Z -201.146,A -90.000,B 90.000,C 0.000} C_DIS
LIN {X -19.732,Y -33.308,Z -198.796,A -90.000,B 90.000,C 0.000} C_DIS
LIN {X -16.359,Y -33.308,Z -196.237,A -90.000,B 90.000,C 0.000} C_DIS
LIN {X -12.970,Y -33.308,Z -193.523,A -90.000,B 90.000,C 0.000} C_DIS
LIN {X -9.451,Y -33.308,Z -190.587,A -90.000,B 90.000,C 0.000} C_DIS
LIN {X -5.708,Y -33.308,Z -187.377,A -90.000,B 90.000,C 0.000} C_DIS
LIN {X -2.584,Y -33.308,Z -184.611,A -90.000,B 90.000,C 0.000} C_DIS
LIN {X -2.022,Y -33.308,Z -184.120,A -90.000,B 90.000,C 0.000} C_DIS
LIN {X 0.630,Y -33.308,Z -181.681,A -90.000,B 90.000,C 0.000} C_DIS
LIN {X 1.405,Y -33.308,Z -180.982,A -90.000,B 90.000,C 0.000} C_DIS
LIN {X 3.856,Y -33.308,Z -178.605,A -90.000,B 90.000,C 0.000} C_DIS
LIN {X 4.624,Y -33.308,Z -177.884,A -90.000,B 90.000,C 0.000} C_DIS
LIN {X 6.836,Y -33.308,Z -175.543,A -90.000,B 90.000,C 0.000} C_DIS
LIN {X 7.167,Y -33.308,Z -175.191,A -90.000,B 90.000,C 0.000} C_DIS
LIN {X 7.517,Y -33.308,Z -174.732,A -90.000,B 90.000,C 0.000} C_DIS
LIN {X 9.191,Y -33.308,Z -172.677,A -90.000,B 90.000,C 0.000} C_DIS
LIN {X 10.269,Y -33.308,Z -170.909,A -90.000,B 90.000,C 0.000} C_DIS
LIN {X 10.609,Y -33.308,Z -170.372,A -90.000,B 90.000,C 0.000} C_DIS
LIN {X 10.678,Y -33.308,Z -170.245,A -90.000,B 90.000,C 0.000} C_DIS
LIN {X 11.573,Y -33.308,Z -167.492,A -90.000,B 90.000,C 0.000} C_DIS
LIN {X 11.642,Y -33.308,Z -166.385,A -90.000,B 90.000,C 0.000} C_DIS
LIN {X 11.591,Y -33.308,Z -165.653,A -90.000,B 90.000,C 0.000} C_DIS
LIN {X 11.587,Y -33.308,Z -165.596,A -90.000,B 90.000,C 0.000} C_DIS
LIN {X 11.565,Y -33.308,Z -165.094,A -90.000,B 90.000,C 0.000} C_DIS
LIN {X 11.342,Y -33.308,Z -163.637,A -90.000,B 90.000,C 0.000} C_DIS
LIN {X 10.947,Y -33.308,Z -162.249,A -90.000,B 90.000,C 0.000} C_DIS
LIN {X 10.900,Y -33.308,Z -162.127,A -90.000,B 90.000,C 0.000} C_DIS
LIN {X 10.258,Y -33.308,Z -160.829,A -90.000,B 90.000,C 0.000} C_DIS
LIN {X 10.020,Y -33.308,Z -160.379,A -90.000,B 90.000,C 0.000} C_DIS
LIN {X 9.016,Y -33.308,Z -159.175,A -90.000,B 90.000,C 0.000} C_DIS
LIN {X 8.734,Y -33.308,Z -158.795,A -90.000,B 90.000,C 0.000} C_DIS
LIN {X 6.822,Y -33.308,Z -157.329,A -90.000,B 90.000,C 0.000} C_DIS
LIN {X 6.671,Y -33.308,Z -157.261,A -90.000,B 90.000,C 0.000} C_DIS
LIN {X 5.915,Y -33.308,Z -156.899,A -90.000,B 90.000,C 0.000} C_DIS
LIN {X 4.520,Y -33.308,Z -156.204,A -90.000,B 90.000,C 0.000} C_DIS
LIN {X 1.169,Y -33.308,Z -155.233,A -90.000,B 90.000,C 0.000} C_DIS
LIN {X 0.812,Y -33.308,Z -155.124,A -90.000,B 90.000,C 0.000} C_DIS
LIN {X 0.702,Y -33.308,Z -155.086,A -90.000,B 90.000,C 0.000} C_DIS
LIN {X 0.289,Y -33.308,Z -155.016,A -90.000,B 90.000,C 0.000} C_DIS
LIN {X -0.111,Y -33.308,Z -154.903,A -90.000,B 90.000,C 0.000} C_DIS
LIN {X -2.506,Y -33.308,Z -154.186,A -90.000,B 90.000,C 0.000} C_DIS
LIN {X -3.578,Y -33.308,Z -153.942,A -90.000,B 90.000,C 0.000} C_DIS
LIN {X -4.018,Y -33.308,Z -153.822,A -90.000,B 90.000,C 0.000} C_DIS
LIN {X -5.796,Y -33.308,Z -153.171,A -90.000,B 90.000,C 0.000} C_DIS
LIN {X -7.652,Y -33.308,Z -152.549,A -90.000,B 90.000,C 0.000} C_DIS
LIN {X -8.086,Y -33.308,Z -152.377,A -90.000,B 90.000,C 0.000} C_DIS
LIN {X -9.547,Y -33.308,Z -151.721,A -90.000,B 90.000,C 0.000} C_DIS
LIN {X -11.593,Y -33.308,Z -150.853,A -90.000,B 90.000,C 0.000} C_DIS
LIN {X -12.019,Y -33.308,Z -150.641,A -90.000,B 90.000,C 0.000} C_DIS
LIN {X -12.334,Y -33.308,Z -150.469,A -90.000,B 90.000,C 0.000} C_DIS
LIN {X -15.597,Y -33.308,Z -148.755,A -90.000,B 90.000,C 0.000} C_DIS
